# B&R Automation Studio project TD52 (part 85)

```iecst
	tLX2_Perm_aux : 	STRUCT
		iFiltConst_LeanoxDev_Gen1 : UINT; (*Filter coefficient PT1 - Leanox deviation for LX2 steady state - Gen1 [sec]*)
		rThreshold_LeanoxDev_Gen1 : REAL; (*Threshold leanox deviation for LX2 steady state - Gen1 [mbar]*)
		rThreshold_Pnorm_LX2_ramp : REAL; (*Threshold norm. power change within 1 second interval for LX2 load ramp detection [0...1]*)
		rThreshold_Pnorm_LX2_step : REAL; (*Threshold norm. power filters difference for LX2 load step detection [0...1]*)
	END_STRUCT;
	tLX2Map : 	STRUCT
		GasType : ARRAY[0..4]OF tLX2_GasType;
	END_STRUCT;
	tLX2_GasType : 	STRUCT
		rLX2_BPOC : ARRAY[0..10]OF REAL; (*actual LX2 BPOC from Permanent Storage [bar]*)
		bLX2_BPOC_measured : ARRAY[0..10]OF BOOL; (*LX2 BPOC - binary map of already measured points [true->measured]*)
	END_STRUCT;
	Pos_WG : 	STRUCT
		Exist : BOOL; (*WG position available (either CAN communication or good quality fo analog input)*)
		Act : REAL; (*WG actual position norm*)
		Set : REAL; (*WG target position norm*)
	END_STRUCT;
	WG_ActuatorState : 	STRUCT
		PosCtrl : USINT := 1; (*Position Control*)
		SelfCal : USINT := 2; (*Self Calibration*)
		Learn : USINT := 3; (*Learn*)
		WipeCycl : USINT := 5; (*Wiping Cycle*)
		Override : USINT := 6; (*Override*)
		ElFailSafe : USINT := 7; (*Electrical Failsafe*)
		ElFailSafeOv : USINT := 8; (*Electrical Failsafe then Override*)
	END_STRUCT;
	WG_StatusMSG : 	STRUCT
		Pos_Act : UINT; (*Actual Shaft Position *)
		T : INT; (*Internal Temperature range: -55 C to +195 C*)
		Pos_Set : UINT; (*Setpoint Position*)
		Fault : USINT; (*Actuator Fault*)
		State : USINT; (*Actuator State*)
		Pos_Set_Norm : REAL; (*Target Position related to Nominal*)
		Pos_Act_Norm : REAL; (*Actual Shaft Position related to Nominal*)
	END_STRUCT;
END_TYPE
```

### Modul_EngCtr.var - Package variables
```iecst
(********************************************************************
 * COPYRIGHT -- INNIO Company
 ********************************************************************
 * Package: Opstate_Pkg
 * File: module_Opstate.typ
 * Author: Mario Graus
 * Created: October 19, 2011
 ********************************************************************
 * Data types of package Opstate_Pkg
 ********************************************************************)
VAR
	IN_EC : IN_EngCtr_Struct;
	OUT_EC : OUT_EngCtr_Struct;
	ParaFactoryDefault : Para_Struct; (*First Init Values*)
	Para : Para_Struct;
	pm : Para_Struct;
	Map : Map_Struct; (* Self learning Data*)
	Cnt : Cnt_Struct; (* Self learning Data*)
	Perm : Perm_Struct; (* Permanent Data*)
	ParaEC : Gtyp_Struct;
	MM2VIS : MM2VIS_Struct;
	VIS2MM : VIS2MM_Struct;
	bEC_Trace_Trigger : BOOL; (* Trigger PV for Traces *)
	iTFilterTVref : UINT;
	iSG_PBC_GlowRed : INT;
	ucGS : USINT; (*Gas Sort (gasart)*)
	xLX2 : fLX2;
	xTrStRed : fTrStRed;
	iCntEC : USINT; (* counter variable reuseable *)
	bWG_CAN_A_Learn_On_Vis : BOOL := 0;	(*Learn On signal to VISU WG A*)
	bWG_CAN_B_Learn_On_Vis : BOOL := 0;	(*Learn On signal to VISU WG B*)
END_VAR
(* IN_EngCtr *)
VAR
	xOpMode : OpMode;
	xEngType : EngType;
	rV_EngDis : REAL; (*Engine Displacement [m3]*)
	rN_Eng : REAL; (*Engine Speed [1/min]*)
	bNewEngCycle : BOOL; (*TRUE = new engine cycle trigger*)
	bType6_Update : BOOL; (* Enables type 6 controls update*)
	bSS_PFPDR : BOOL; (* Steady State for PFPDR *)
	bSS_Opt : BOOL; (* Steady State for Optimizer*)
	bSS_LamLim : BOOL; (* Steady State for Lambda Limit*)
	bSS_WG : BOOL; (* Steady State for wastegate *)
	rH_Amb : REAL; (* Sealevel [m] *)
	rPr_Amb : REAL; (* Ambient pressure [bar] *)
	bWasActivatedGen2Idle : BOOL := FALSE;
	bIsActiveGen2Idle : BOOL := FALSE;
	rVE_Eng : REAL; (* Volumetric Efficiency *) (* OldName: rLieferGMotor; Cycle: 2 *)
	rLam_PI : REAL; (* lambda for port injection opening duration calculation *)
	xGridStat : fGridStat;
	rN_Set_Norm : REAL := 1.0; (*Speed setpoint normalized for Engine Controller*)
END_VAR
(* misf_ctr *)
VAR
	bTrip_Misf : BOOL; (* Trip: A1047 Misfiring failure *) (* OldName: AUSS_A; Cycle: 2 *)
	bWarn_Misf : BOOL; (* Warning: W3217 Misfiring failure *)
	bMisfBlink : BOOL;
	iCnt_Misf : USINT;
END_VAR
(* IgnPoint *)
VAR
	rCA_IP_Set : REAL; (* actual ignition timing setpoint *) (* OldName: W_ZZP; Cycle: 2 *)
	bSG_PBC_GlowRed : BOOL; (*Release FPR/SCO through PBC*) (* OldName: bReductionGlow_Pi; *)
	bPBC_IPRed : BOOL; (*Betriebsmeldung ZZP-Reduktion Gluehzuenden / Pmax*) (* OldName: bZZPRed_DMR; *)
	iPBC_IPRed : USINT; (*Betriebsmeldung ZZP-Reduktion Gluehzuenden / Pmax*) (* OldName: ucDMRZZPRed; *)
	iCyl_IP_Act_Min : USINT; (*Nummer vom Zylinder mit kleinsten ZZP*)
	bTrStRed_Running : BOOL; (* TrStRed function running status *)
	bTrStRed_hiEGT_dis : BOOL; (* high avg.EGT pw.red. disable / timer extension for high cyl.max.EGT alarm by TrStRed function *)
	bTrStRed_SteadyState_Loss_LX2 : BOOL; (* Leanox plus steady state loss by TrStRed function *)
	bMsg_TrStRed_Start : BOOL; (* TrStRed function cycle started - operator message *)
	bMsg_TrStRed_Complete : BOOL; (* TrStRed function cycle completed - operator message *)
	rCA_IPOffs_SCRInTemp : REAL;
END_VAR
(* dyn_GR *)
VAR
	bBM_GrC_Event : BOOL; (* Low Voltage Ride Through Event *)
	bBM_PoleSlip : BOOL; (* Mains failure + Generator Pole slip *)
	bBM_Disc_dynAng : BOOL; (* Mains failure + dynamic rotor angle maximum *)
	bBM_Disc_staticAng : BOOL; (* Mains failure + static rotor angle maximum*)
	bBM_Disc_CapMode : BOOL; (* Mains failure + leading power factor operation *)
	bBM_Disc_dynAng_Min : BOOL; (* Mains failure + dynamic rotor angle minimum *)
	bBM_Disc_Power : BOOL; (* Mains failure + electric power to low *)
	bBM_FRT_Event : BOOL; (* Fault Ride Through Event in island operation *)
	bBM_PoleSlip_EPS : BOOL; (* Generator Pole slip in island operation *)
	bBM_GrC_Event_Sim : BOOL; (* Low Voltage Ride Through Event simulated *)
	bGC_LeanoxErr_AUS : BOOL := FALSE; (*TRUE = Stoerung A1080 deaktiviert ueber GCEvent*)
	iMissfCyl_GrC : UDINT; (* 0 *) (* OldName: MissfCyl_GC; Cycle:2; *)
	bGrC_PowerFIX_HVRT : BOOL; (* TRUE = Leistungsfixierung im eng_ctr aktiv (Zeit laeuft) --> HVRT Event*) (* OldName: bGC_PowerFIX; Cycle:2; *)
	bGrC_PowerFIX : BOOL; (* TRUE = Leistungsfixierung im eng_ctr aktiv (Zeit laeuft) --> LVRT Event*) (* OldName: bGC_PowerFIX; Cycle:2; *)
	bGC_maintenance_request : BOOL; (* Mains failure maintenance request *) (* OldName: bGC_maintenance_request ; Cycle:2; *)
	bGrC_TCPumpAkt : BOOL; (* TRUE=Pumperkennung aus dyn. GC aktiv fuer gas_flow *) (* OldName: bGC_TCPumpAkt; Cycle:2; *)
	bGrC_LambAdabtAKT : BOOL; (* TURE = Lambdaadaption from dyn. GridCode aktiv *) (* OldName: bGC_LambdaAdabtAKT; Cycle:2; *)
	bVoltageLow_cust_OP_MSG : BOOL;
	bGrC_FixActuators : BOOL;
	rPos_WG_GrC : REAL;
	rPos_CBV_GrC : REAL;
	bIgnOffTestMode : BOOL := FALSE; (*TRUE = Zuendung EIN/AUS nach Muster*)
	bIGTLatePhase2ON : BOOL; (*ZZP auf spaet stellen in Phase 2 JA/NEIN*)
	bIGTLatePhase2 : BOOL; (*Befehl an ignpoint Task - ZZP auf spaet stellen*)
	rCA_Ign_Act_late_GC : REAL; (*[deg CA] spaeter ZZP fuer Phase 2 von IGNTestMode (GridCode)*)
	bFreeze_GEN2 : BOOL;
	rPos_CBV_Freeze : REAL;
	rPos_TV_Freeze : REAL;
	rPos_WG_Freeze : REAL;
	rGrid_OffsetFactor : REAL; (* PI-Duration offset from dynamic gridcode *)
	rGasflow_Factor_GrC : REAL; (* Gasflow factor from dynamic gridcode *)
	bGrC_GCB_DCON_FRT : BOOL; (* Open signal to GCB due to pole slip *)
	bGrC_GCB_DCON_FRT_EPS : BOOL; (* Open signal to GCB due to pole slip in island operation *)
	bLeanox_Man_old_FRT : BOOL; (* LEANOX controller status before FRT event *)
END_VAR
(* GR_GCB_cust *)
VAR
	bF_UnderMp_Lo : BOOL; (* W9312: Generator frequency too low in mains parallel operation *)
	bF_OverMp_Hi : BOOL; (* W9313: Generator frequency too high in mains parallel operation *)
	iTFilt_N_GR : UINT := 2000;
	rN_GR_Filt : REAL; (* Filtered engine speed for LEANOX speed compensation *)
	rF_GR_Filt : REAL; (* Filtered engine frequency for ITP reduction *)
END_VAR
(* GAS FLOW *)
VAR
	rP_Rot : REAL; (*Rotationsleistung in [kW]*)
	rLam_Trans_Corr : REAL; (*transient Lambda correction*)
	TJ_GASO : BOOL;
	TJ_GASO_B : BOOL;
	ucTJ_GASO : USINT;
	TJ_GASM : BOOL;
	TJ_GASM_B : BOOL;
	ucTJ_GASM : USINT;
	rFlow_TV_x : REAL; (*LIVC actual Volumeflow for TV Controller*)
	rFlow_TV_w : REAL; (*LIVC setpoint Volumeflow for TV Controller*)
	rFlow_CBV_x : REAL; (*LIVC actual Volumeflow for CBV Controller*)
	rFlow_CBV_w : REAL; (*LIVC setpoint Volumeflow for CBV Controller*)
	bBM2852_PumpPuls : BOOL; (*B2852 - Turbolader Pumpen*)
	rLam_TJ_Set : REAL; (* Lambda for TecJet *)
	rPr_P2s_df : REAL; (*P2s Digital gefiltert in [bar]*)
	rPr_P2s_df_TJ : REAL; (*P2s Digital gefiltert in [bar]*)
	rCBV_CDS_Speed_D_Offset : REAL; (*T6 GEN1 CBV derivative gain scheduling*)
	rTV_CDS_Speed_D_Offset : REAL; (*T6 GEN1 TV derivative gain scheduling*)
END_VAR
(* LEANOX *)
VAR
	rP_Act_l : REAL;
	rPr_Leanox_Set : REAL; (* Setpoint boost pressure *) (* Oldname: pl_soll; Cycle: 2*)
	rLam_Leanox_Set : REAL; (* Setpoint lambda *) (* Oldname: OUT_EC.rLam_Eng_LL_Set; Cycle: 2*)
	RPSW3 : BOOL; (*Warning: LEANOX algorithm failure*)
	RPSA7 : BOOL;
	rPr_CH_PFPDR_Calc : REAL; (* Boost pressure offset calculated for PFPDR*)
	rNum_ConvLamtoP2s : REAL := 2; (* Conversion rate from lambda to boost pressure for PFPDR*)
	rPr_CH_PFPDR_Offs : REAL; (* Boost pressure offset from PFPDR to Gen2 controller*)
	rCorr_LX_GR : REAL; (* Speed compensation factor for LEANOX *)
	rPr_Leanox_Offs_H2 : REAL; (* Boost pressure offset H2 content [bar] *)
END_VAR
(* eng_ctr *)
VAR
	rPos_TV_u : REAL; (*Regler Ausgang ohne skalierung*)
	iMisfCyl_OverSpeed : UDINT; (*ACHTUNG hier braucht es noch Klaerung*)
	bLR_IGN_Retard : BOOL; (*retard ignition timing point to react on a load rejection by the GCB*)
	pm_stat_var_LR : ARRAY[0..100] OF tStat_VAR_LR := [101(0)]; (*statistic structure to save the speed gradient values at engine shut down with time stamps*)
	pm_stat_var : ARRAY[0..100] OF tStat_VAR := [101((0))]; (*statistic structure to save the speed gradient values at engine shut down with time stamps*)
	iCounter_stat_var_LR : INT := 0;
	iCounter_stat_var : INT := 0; (*counter and index variable for statistic structure for the speed gradient values*)
	rN_LR_IGN_Retard_HOLD : REAL := 1.1; (*Speed threshold to keep ITP retard during LR [p.u.]*)
	rTi_LR_GasStop_largeRej : REAL := 0.4; (*Duration of gas-stop for big load rejections [s]*)
	rTi_LR_GasStop_smallRej : REAL := 0.1; (*Duration of gas-stop for small load rejections [s]*)
END_VAR
(* Msg EC *)
VAR
	bGnlTrip : BOOL;
	bGnlTrip1 : BOOL;
	bGnlTrip2 : BOOL;
	bGnlTrip3 : BOOL;
	bGnlWarning : BOOL;
	AmmSeq_PiPosAbw : AmmSequence; (* Trip: W2470, OM: B2929 *) (* Oldname: AmmSeq_PiPosAbw *)
END_VAR
(* gen_EC_T2 *)
VAR
	bAct_Mon_Release : BOOL; (*Throttle valve failure monitoring release*)
	bAct_Mon_Rel_WG : BOOL; (*Release monitoring for wastegate actuator*)
	tDataRec_EEPROM : ARRAY[0..7] OF BYTE := [8(0)]; (*CAN wastegate read data A - 8 bytes*)
	tDataRec_EEPROM_Info : ARRAY[0..7] OF BYTE := [8(0)]; (*CAN wastegate read data A - 8 bytes*)
	tCAN_WG_ADDR_A : BYTE := 0; (*CAN wastegate A source address*)
	tCAN_WG_ADDR_B : BYTE := 0; (*CAN wastegate B source address*)
	tNewADDR : BYTE := 0; (*CAN wastegate new address to configure EEPROM*)
	tWG_CAN_B_ActSrcAdd : BYTE := 0; (*CAN wastegate actuator B source address*)
	tWG_CAN_A_ActSrcAdd : BYTE := 0; (*CAN wastegate actuator A source address*)
END_VAR
(* parEC *)
VAR
	bNoInitDetected : BOOL := FALSE; (*allways true, except 1cycle on init up*)
END_VAR
(* hum_pac_EC *)
VAR
	rpl_soll_Max_filt : REAL;
	rpl_ist_filt : REAL;
	AbsHumidity : REAL; (* absolute humidity air intake [g/kg] *)
	bMsg_Hum_T2sOffs_Act : BOOL;
	bMsg_Hum_Pred_Lim : BOOL;
	pbaro : REAL; (* barometric pressure used for humidity control [bar] *)
	rP2s_Comp_HumOffset : REAL; (* [bar] *)
	rT_T2_HumOffset : REAL; (*  *)
	rMassFlow_Gas : REAL; (* gas mass flow [kg_gas/h] *)
	rMassFlow_AirIn : REAL; (* intake air mass flow [kg_air/h] *)
	AbsHumidity_Mixture : REAL; (* absolute humidity mixture [kg_H2O/kg_mix] *)
	rGasFlowN : ARRAY[0..4] OF REAL; (* gas flow [m^3/h] *)
	bHum_GasIn_Abs_MSF : BOOL; (* measuring signal failure customer signal BUS *)
	AbsHumidity_AirIn : REAL; (* absolute humidity air intake [g/kg] *)
	AbsHumidity_Mix : REAL; (* absolute humidity mixture [g/kg] *)
END_VAR
(* Exhaust *)
VAR
	AN_ABMWN : ARRAY[0..25] OF BOOL; (* Koppelfeld Abweichung neg vom Mitt*)
	AN_ABMWN_B : BOOL; (* dev. exh. avg. operating message *)
	AN_ABMWN_W : BOOL; (* negative dev. exh. avg. warning *)
	AN_ABMWP : ARRAY[0..25] OF BOOL; (* Koppelfeld Abweichung pos vom Mitt*)
	AN_ABMWP_B : BOOL; (* dev. exh. avg. operating message *)
	AN_ABMWP_W : BOOL; (* positive dev. exh. avg. warning *)
	AN_ATMA : BOOL;
	bZylAusfall : BOOL;
	bMsg1049_Test : BOOL;
	MS_AGT : BOOL;
	MSAGT : ARRAY[0..25] OF BOOL;
	MSAGT_W : BOOL;
	t_zyl : ARRAY[0..25] OF INT;
	bSCO_EGT_DltLim : BOOL; (* - *) (* OldName: AGT_DELTA; *)
	iNum_Cyl_EGT_Max : USINT; (*Hottest cylinder number*) (* OldName: ucZYL_MAX_Cyl; *)
	AN_ABMW : BOOL;
	AN_ATM : ARRAY[0..25] OF BOOL;
	MSAGT_B : BOOL;
	AN_ATMA_B : BOOL;
	rT_EG_MaxLim : REAL; (*exhaust gas temperature maximum limit*)
	xTExhMon : fTExhMon := (0); (*FuB*)
	bMsg2339_Set : BOOL; (* A2339: Exhaust gas temperature inclination maximum at cylinder head *)
	bMsg2970_Set : BOOL; (* B2970: Exhaust gas temperature inclination maximum at cylinder head *)
	iNum_Msg2970 : USINT;
	bHoldBackfPrev : BOOL;
	bMsg9388_Set : BOOL; (*W9388: Combustion anomaly detected*)
	bMsg9092_Set : BOOL; (*B9092: Combustion anomaly detected*)
END_VAR
(* GLOW IGN *)
VAR
	bSG_TV : BOOL; (*Enables TV alternation by GlowIgnition Task*)
	rPos_SG_TV : REAL; (*alternated TV postion*)
	bSG_CBV : BOOL; (*Enables CBV alternation by GlowIgnition Task*)
	rPos_SG_CBV : REAL; (*alternated CBV position*)
	bSG_Rel_Mon : BOOL; (* monitoring release for special gas applikation *) (* Oldname: FG_TS_UW *)
	bSCO_BLOCK1 : BOOL; (* Blockierung Sicherheitsschliessen *) (* OldName: SS_BLOCK1; *)
	bSCO_BLOCK2 : BOOL; (* Blockierung Sicherheitsschliessen *) (* OldName: SS_BLOCK2; *)
	bSG_PBC_GlowIgnFailure : BOOL; (* Glow ignition failure by PBC *) (* OldName: bDMR_A_GLOW; *)
	rSG_GasLimit : REAL; (* special gas factor for gasflow limit *) (* OldName: ssGasLimit; *)
	bSG_BackFireDetection : BOOL; (* Trip A2283 *)
	bSG_TV_FGQC : BOOL; (* Fix TV position *)
	bSG_CBV_FGQC : BOOL; (* Fix CBV position *)
	rPos_SG_TV_FGQC : REAL; (* TV position FGCQ *)
	rPos_SG_CBV_FGQC : REAL; (* CBV position FGCQ *)
	b2975_Set : BOOL; (* Operation message 2975 *)
	bFGQC_Active : BOOL; (* Fast gas quality change function active *)
	bLeanox_Man_oldFGQC : BOOL; (* LEANOX controller status before FGQC event *)
	bFPR_Active : BOOL; (* Fast power reduction function active *)
	bLeanox_Man_old_FPR : BOOL; (* LEANOX controller status before FPT event *)
END_VAR
(* PFPDR *)
VAR
	rLam_PFPDR_Offs : REAL; (* Lambda Offset during PFPDR *)
	bPFPDR_IPCorr_dis : BOOL; (* disables IP correction during PFPDR *)
	rCA_IP_PFPDR_Offs : REAL;
	bPFPDR_CylOpt_dis : BOOL;
	bPFPDR_CBVOpt_dis : BOOL;
	bPFPDR_Act : BOOL;
	bIP_CBVOpt : BOOL; (* CBVOpt aktiv? *)
	rCA_IP_PFPDR_Prof : ARRAY[0..24] OF REAL;
	MFB50Ctr : AI50toIT;
	bTrace_var : BOOL := 0;
	rCA_MFB50_Filt_type9 : ARRAY[0..24] OF REAL;
	rCA_MFB50_Filt_type6_Max : REAL;
	rCA_MFB50_Filt_type6_Min : REAL;
	rCA_MFB50_Filt_type6_Avg : REAL;
	rCA_MFB50_Filt_type6 : ARRAY[0..24] OF REAL;
	rCA_MFB50_Filt_type6_Median : REAL;
	rCA_MFB50_Filt_type9_Median : REAL;
	rCA_MFB50_type9_Set : REAL;
	rCA_MFB50_Filt_type9_Min : REAL;
	rCA_MFB50_Filt_type9_Max : REAL;
	rCA_MFB50_Filt_type9_Avg : REAL;
	rCA_MFB50_type6_Set : REAL;
	rPr_Leanox_Offset_CoV : REAL;
	rPos_TB34_SG : REAL;
	iTB34CtrMode : INT;
	bTrip_LambdaLimit : BOOL; (*A2294: Lambda limit exceeded*)
	bMsg_p2soutofRange : BOOL; (*B2897: Boost pressure out of range*)
	bGEN2_Block_P2_Err : BOOL; (* Block Gen2: no P2 pressure signal available *)
	xGen2 : Gen2;
	bGEN2_FDC_active : BOOL; (*Activate Hangs FDC in GEN2 control*)
	bVerrigelung_EXHT : BOOL;
	refPoint_Lambda_start : ARRAY[0..9] OF lcrCurveByPoints_TabEntry_type;
	LCRCByP_Lambda_start : LCRCurveByPoints;
	refPoint_ITP : ARRAY[0..9] OF lcrCurveByPoints_TabEntry_type;
	LCRCByP_ITP : LCRCurveByPoints;
	refPoint_LamLoLim_coldFS_ABS : ARRAY[0..9] OF lcrCurveByPoints_TabEntry_type; (* y = abs lam limit and x = pressure in [bar] *)
	refPoint_LamLoLim_ABS : ARRAY[0..9] OF lcrCurveByPoints_TabEntry_type; (* y = abs lam limit and x = pressure in [bar] *)
	refPoint_LamUpLim_ABS : ARRAY[0..9] OF lcrCurveByPoints_TabEntry_type; (* y = abs upper lam limit and x = pressure in [bar] *)
	rZZPStart_T4_low : REAL;
	rZZPStart_T4_high : REAL;
	bITPStTEMP : BOOL;
	bFirstStepAct : BOOL;
	bExhTempDep : BOOL;
	rFirstStepITPOffs : REAL;
	rSecondStepITPOffs : REAL;
	rCA_IT_GEN2_FS_rel : REAL;
	ulGasFlow_M_FDC : UDINT; (*[Nl/s] * 1000*)
	ulGasFlow_FDC : UDINT; (*[Nl/s] * 1000*)
	rN_StartITOffs_full : REAL;
	rN_StartITOffs_zero : REAL;
	rCA_IP_Set_Raw_GEN2_FS : REAL;
	rP_IT_FS_LimNorm : REAL;
	tmaxITP : TIME;
	rCA_IT_Offs_Start : REAL;
	rCA_IP_Gen2_Offs : REAL;
	rCA_IP_Gen2_NetP_Offs : REAL;
	bGEN2_FS_IP_Set : BOOL := 0;
	rZZPStart_Tcyl_low : REAL := 0;
	rZZPStart_Tcyl_high : REAL := 0;
	rCA_IP_Set_Raw_normal : REAL;
	rT_EG_H : ARRAY[0..24] OF REAL;
	TP_10ms_OptiChng : TP_10ms := (0);
	iCount_steady : INT;
	iNum_steady_state : INT;
	bdeltaPr_TV_actuateTV : BOOL;
	rGainTV_rDeltaPr_TV : REAL;
	rDeltaPr_TV_integrator_TV : REAL;
	rDeltaPr_TV_integrate_TV_ON : REAL;
	rPr_CBV_Release : REAL;
	rPr_CBV_Lock : REAL;
	deltaPr_TV_ref_data : ARRAY[0..5] OF lcrCurveByPoints_TabEntry_type;
	deltaPr_TV_CBV_gain_data : ARRAY[0..5] OF lcrCurveByPoints_TabEntry_type;
	deltaPr_TV_TV_gain_data : ARRAY[0..5] OF lcrCurveByPoints_TabEntry_type;
	CBV_lim_byTV_data : ARRAY[0..4] OF lcrCurveByPoints_TabEntry_type;
	LCRCurve_TV_min_table : ARRAY[0..7] OF lcrCurveByPoints_TabEntry_type;
	LCRCurve_TV_min_CBV_table : ARRAY[0..2] OF lcrCurveByPoints_TabEntry_type;
	rP_LR_Trig_ActSat_CBV : REAL;
	rTi_LR_ActSat_CBV : REAL;
	xLCRCurve_R_Rot_Correction_data : ARRAY[0..8] OF lcrCurveByPoints_TabEntry_type;
	rDelta_a_red : REAL := 0.0;
	bSIMPID_EXT_TV_Act : BOOL := FALSE;
	bSIMPID_EXTERN_AW_TV : BOOL := FALSE;
	bSIMPID_EXTERN_AW_CBV : BOOL := FALSE;
	bSTOPint_cbv_trans : BOOL := FALSE;
	rP_el_LockTV_Norm : REAL; (*Power trigger value to lock the throttle valve in island mode in upper load range*)
	rP_el_ReleaseTV_Norm : REAL; (*Power trigger value to release the throttle valve in island mode*)
	tTimeTrigger : TIME := T#150ms;
	tTimeTrigger_HiGasDens : TIME := T#60ms;
	ulGasSprungVol : UDINT; (*[l/s]*1000*)
	ulGasSprungVol_HiGasDens : UDINT; (*[l/s]*1000*)
	bstveract : BOOL;
	bGasSprung : BOOL;
	ulatvergasvol : UDINT;
	ulGasSprungMax : UDINT; (*[l/s]*1000*)
	iGasSprungThresh_HiGasDens : INT; (*[g/Nm3]*)
	bUseTVIdleControl : BOOL; (*TRUE = Engine uses TV control without skipfire for engine start and idle control*)
	rKp_Gen2SkipF_Pnom : REAL;
	rKp_Gen2SkipF_Pskip : REAL;
	rP_LimitBDCCBV_ff_Active : REAL;
END_VAR
(*LeanoxDrift*)
VAR
	bWarn_Nox_Meas_recommend : BOOL; (*warning for recommend leanox adjustment*)
	bWarn_Nox_Meas_mandatory : BOOL; (*warning for mandatory leanox adjustment*)
	bMsg_B2937 : BOOL; (*B2937: operating message for performed leanox adjustment*)
	bMsg_B2938 : BOOL; (*B2938: operating message for performed combustion chamber cleaning*)
	bCBV_closed_Start_SY : BOOL; (*TRUE = CBV closed at engine start until SY*)
	bParaSetupOk_10s : BOOL; (*Para Setup OK + 10sec*)
	bFS_Ramp_Rel : BOOL;
	bTiStart5min_Ena : BOOL;
	bEngine_was_stopped : BOOL := 0;
	rF_LEANOX_Err : REAL := 1.0;
	bGEN2_RAMP_ACTIVE : BOOL := 0;
	bUseColdFS_LamLim : BOOL := 0; (*Use cold Fast Start low Lambda Limits for GEN2*)
	bMisfGEN2 : BOOL := TRUE; (*activate misfire computed from GEN2 control*)
	iMissfCyl_GEN2 : UDINT := 0; (*number of skipped cylinders from GEN2 control*)
	refPoint_addKpLam_Kp_y : ARRAY[0..5] OF REAL; (*reference add Lambda Kp GEN2 island*)
	rKeAdaptRL : REAL; (*reference gain for adaption GEN2 island*)
	rKeAdaptGain : REAL; (*reference rate limit for adaption GEN2 island*)
	rITCtransDeltaAcc_y : ARRAY[0..4] OF REAL; (*reference for transient ignitioin timing point change of GEN2 to avoid knocking*)
	refPoint_iLQR_Q0_y : ARRAY[0..5] OF REAL; (*reference Q0 GEN2 island*)
	refPoint_addKpLam_Ti_y : ARRAY[0..5] OF REAL; (*reference add Lambda Ti GEN2 island*)
	refPoint_iLQR_Keng_y_pow : ARRAY[0..6] OF REAL; (*reference to reset learning function*)
	refPoint_iLQR_Keng_y : ARRAY[0..12] OF REAL; (*reference to reset learning function*)
	bdcCbv_rKp_island_Lup : ARRAY[0..9] OF REAL; (*reference gain scheduling Kp bypass valve for GEN2 BDC island*)
	bdcTv_rKp_island_Lup : ARRAY[0..9] OF REAL; (*reference gain scheduling Kp throttle valve for GEN2 BDC island*)
	refPoint_iLQR_R1_y : ARRAY[0..5] OF REAL; (*reference R1 GEN2 island*)
	bAutoLoad_Island : BOOL; (*Werte fuer GEN2 Inselbetrieb laden in PV-CHECK*)
END_VAR
(* ESC *)
VAR
	rLamLimOffs_ESC : REAL; (* Lambda lower limit offset ESC *)
	rP_Ramp_IncGrad_Offs_ESC : REAL; (* Power ramp offset ESC *)
END_VAR
(*Leanox 2.0*)
VAR
	bLX2_active : BOOL; (*Leanox 2.0 active [true->active]*)
	bWarn_LX2_inLimit : BOOL; (*Leanox 2 saturation - warning*)
	bMsg_LX2_Active : BOOL; (*Leanox 2 Active - operator message*)
	bMsg_LX2_NotActive : BOOL; (*Leanox 2 Not Active - operator message*)
	bMsg_LX2_MapReset : BOOL; (*Leanox 2 Map Reset Request from HMI - operator message*)
	rMFIntOutMax : REAL; (*Misfire level used for ESC and LX2*)
	rPr_LX2_offset : REAL; (* Leanox 2.0 boost pressure offset *)
	rGain_ss_boost_iLQR : REAL := 0.0;
	rGain_ss_boost_iLQR_OUT : REAL := 0.0;
	bDemPermSave : BOOL;
END_VAR
(* FastStart *)
VAR
	bLoad_reached : BOOL;
	bTarLoad_reached : BOOL;
	bTarLoad_blockOM : BOOL;
	xTP_TarLoad_reached : TP;
	bFS_Island_Ena : BOOL; (* island fast start enabled *)
END_VAR
(* Direct Air Injection *)
VAR
	xDAI : fDAI; (* direct air injection FB *)
	bDAI_MSF : BOOL; (* direct air injection measuring signal failure *)
	bDAI_V_Close_Fault : BOOL; (* direct air injection shut off valve closing fault *)
	bDAI_V_Open_Fault : BOOL; (* direct air injection shut off valve opening fault *)
	bDAI_Pr_In_Hi : BOOL; (* direct air injection pressure before shut off valve high *)
	TOF_MissfCmd : TOF;
END_VAR
(* TC1 SPP *)
VAR
	rPr_EGbHP_TC1 : tBank_AB; (* P3 Filt TC1*)
	rPr_EGbHP_TC1_UF : REAL;
END_VAR
(* TC2 SPP_EC *)
VAR
	bT_SCR_OXI_TC_valid : BOOL; (*Inlet temperature sensor exist and good quality - SCR in, SCR out, OXIcat In, Turbocharger Out*)
	rT_SCR_OXI_TC_In_Hi : REAL; (*Inlet temperature maximum - SCR in, SCR out, OXIcat In, Turbocharger Out [degC]*)
END_VAR
(* Wastegate *)
VAR
	rPos_CBV_Ref_WG : REAL; (*setpoint of position compressor bypass valve for wastegate control*)
	rPosWG_Factor : REAL := 0.0; (*CAN wastegate read position factor*)
	tDataSend_WG : ARRAY[0..7] OF BYTE := [8(0)]; (*CAN wastegate data to send - 8 bytes*)
	iDataSend_WG_Tmp : UINT := 0; (*CAN wastegate set position to be sent - TEMPORARY*)
	tDataSend_WG_Tmp : ARRAY[0..1] OF BYTE := [2(0)]; (*CAN wastegate actuator command TEMPORARY byte*)
	iCAN_WG_B_StatID : ARRAY[0..5] OF UDINT := [6(0)]; (*CAN wastegate actuator B - Actuator Status MSG ID*)
	iCAN_WG_B_ErrID : ARRAY[0..5] OF UDINT := [6(0)]; (*CAN wastegate actuator B - Failures and Warning MSG ID*)
	iCAN_WG_B_SendID : ARRAY[0..5] OF UDINT := [6(0)]; (*CAN wastegate actuator B - Actuator Command MSG ID*)
	iCAN_WG_A_StatID : ARRAY[0..5] OF UDINT := [6(0)]; (*CAN wastegate actuator A - Actuator Status MSG ID*)
	iCAN_WG_A_ErrID : ARRAY[0..5] OF UDINT := [6(0)]; (*CAN wastegate actuator A - Failures and Warning MSG ID*)
	iCAN_WG_A_SendID : ARRAY[0..5] OF UDINT := [6(0)]; (*CAN wastegate actuator A - Actuator Command MSG ID*)
	iCAN_WG_A_T2AID : ARRAY[0..5] OF UDINT := [6(0)]; (*CAN wastegate actuator A - Tool to Actuator MSG ID*)
	iCAN_WG_A_A2TID : ARRAY[0..5] OF UDINT := [6(0)]; (*CAN wastegate actuator A - Actuator to Tool  MSG ID*)
	iCAN_WG_B_T2AID : ARRAY[0..5] OF UDINT := [6(0)]; (*CAN wastegate actuator B - Tool to Actuator MSG ID*)
	iCAN_WG_B_A2TID : ARRAY[0..5] OF UDINT := [6(0)]; (*CAN wastegate actuator B - Actuator to Tool  MSG ID*)
	iCAN_WG_DataLength : ARRAY[0..5] OF USINT := [6(0)]; (*CAN wastegate data length (K_S: 8 bytes)*)
	xCANread_WG_B_EE : CANread := (0); (*CAN wastegate B read function*)
	xCANread_WG_A_EE : CANread := (0); (*CAN wastegate A read function*)
	xCANwrite_WG_B_EE : CANwrite := (0); (*CAN wastegate B write function*)
	xCANwrite_WG_A_EE : CANwrite := (0); (*CAN wastegate A write function*)
	xCANreadID_WG : CANread := (0); (*CAN wastegate A/B ID read function*)
	xCANwrite_WG_B : CANwrite := (0); (*CAN wastegate B write function*)
	xCANwrite_WG_A : CANwrite := (0); (*CAN wastegate A write function*)
	xCANwriteID_WG_B : CANwrite := (0); (*CAN wastegate B write function*)
	xCANwriteID_WG_A : CANwrite := (0); (*CAN wastegate A write function*)
	xCANread_WG_B : CANread := (0); (*CAN wastegate B read function*)
	xCANread_WG_A : CANread := (0); (*CAN wastegate A read function*)
	iWG_CAN_A_State : USINT := 0; (*CAN wastegate actuator A commanded state*)
	iWG_CAN_B_State : USINT := 0; (*CAN wastegate actuator B commanded state*)
	tPos_WG_A : Pos_WG := (0); (*Wastegate position actuator A*)
	tPos_WG_B : Pos_WG := (0); (*Wastegate position actuator B*)
	tPos_WG : Pos_WG := (0); (*Wastegate position actuator single*)
	bActuator_WG_A_Exist : BOOL := FALSE; (*Wastegate actuator A exists*)
	bActuator_WG_B_Exist : BOOL := FALSE; (*Wastegate actuator B exists*)
	bActuator_WG_Exist : BOOL := FALSE; (*Wastegate actuator single exists*)
	bActuator_WG_A_Ok : BOOL := FALSE; (*Wastegate actuator A is OK*)
	bActuator_WG_B_Ok : BOOL := FALSE; (*Wastegate actuator B is OK*)
	bActuator_WG_Ok : BOOL := FALSE; (*Wastegate actuator single *)
	tWG_CAN_A_Warn : ARRAY[0..1] OF BYTE := [2(0)]; (*CAN wastegate A System Warnings*)
	tWG_CAN_A_Fail : BYTE := 0; (*CAN wastegate A Actuator Failures*)
	tWG_CAN_B_Warn : ARRAY[0..1] OF BYTE := [2(0)]; (*CAN wastegate B System Warnings*)
	tWG_CAN_B_Fail : BYTE := 0; (*CAN wastegate B Actuator Failures*)
	bErr_WG_CANcomm_A : BOOL := 0; (*CAN wastegate A CAN communication A2384 set*)
	bErr_WG_CANfail_A : BOOL := 0; (*CAN wastegate A CAN failures W2380 set*)
	bErr_WG_CANwarn_A : BOOL := 0; (*CAN wastegate A CAN warnings W2382 set*)
	bErr_WG_CANcomm_B : BOOL := 0; (*CAN wastegate B CAN communication A2385 set*)
	bErr_WG_CANfail_B : BOOL := 0; (*CAN wastegate B CAN failures W2381 set*)
	bErr_WG_CANwarn_B : BOOL := 0; (*CAN wastegate B CAN warnings W2383 set*)
END_VAR
VAR CONSTANT
	tWG_ActuatorState : WG_ActuatorState := (PosCtrl:=1,SelfCal:=2,Learn:=3,WipeCycl:=5,Override:=6,ElFailSafe:=7,ElFailSafeOv:=8); (*CAN wastegate actuator K&S: available commanded states*)
END_VAR
VAR
	tWG_A_Status : WG_StatusMSG; (*CAN wastegate A CAN Status Information*)
	tWG_B_Status : WG_StatusMSG; (*CAN wastegate B CAN Status Information*)
	bCANread_WG_A_Err : BOOL; (*CAN wastegate A CAN read error trigger bit*)
	bCANread_WG_B_Err : BOOL; (*CAN wastegate B CAN read error trigger bit*)
END_VAR
(* PCGV Monitoring *)
VAR
	xPCGVmon : fPCGVmon; (*FuB PCGV monitoring*)
END_VAR
(* FastSync *)
VAR
	xFSyPrM : fFSyPrM; (* FastSync controller for premixed engines *)
	rPos_TV_FSyOffset : REAL := 0.02; (*TV offset when FastSync controller (premixed) is active*)
	rLam_FSyPrM_Offset : REAL := 0.0; (*Lambda offset by FastSync controller for premixed engines*)
	bFSync_StartFrom0rpm : BOOL := FALSE; (* Fast-sync w. PI: release FastSync controller only at first synchronization, engine starting from standstill*)
	bFSyPrM_StartFrom0rpm : BOOL := FALSE; (* Fast-sync premixed: release FastSync controller only at first synchronization, engine starting from standstill*)
END_VAR
(* Gen2_xt *)
VAR
	refPoint_rEtaBrakeExt : ARRAY[0..5] OF lcrCurveByPoints_TabEntry_type;
	refPoint_rGain_iLQR_rR0 : ARRAY[0..1] OF lcrCurveByPoints_TabEntry_type; (* gain for R0 value *)
	rR0_iLQR : LREAL; (*iLQR spur of R matrix *)
	rPrR_deltaP_TV_x_2 : REAL;
	rPrP2s_GEN2GQCOffs_maxLoLoad : REAL; (*[mbar] maximum GEN2 gasquality change boost pressure offset w/o scaling Parameter*)
	rR_iLQR_0 : REAL := 5.0; (* GEN2 island T6PreM *)
	rR_iLQR_1 : REAL := 40.0; (* GEN2 island T6PreM *)
	rR_iLQR_2 : REAL := 1000000000; (* GEN2 island T6PreM *)
	rR_iLQR_3 : REAL := 1000000000; (* GEN2 island T6PreM *)
	rQ_iLQR_0 : REAL := 1.0; (* GEN2 island T6PreM *)
	rQ_iLQR_1 : REAL := 0.1; (* GEN2 island T6PreM *)
	rQ_iLQR_2 : REAL := 0.0001; (* GEN2 island T6PreM *)
	rP_1_SkipF_Fact : REAL; (* Factor for 0 cylinder skipping power threshold [%Pnom] *)
	refPoint_SkipFLevel : ARRAY[0..4] OF lcrCurveByPoints_TabEntry_type; (* scaling of skip fire level over boost pressure *)
	rQ_KF_3_init : REAL := 0.01;
	rN_ssTVdpCtrl_0 : REAL := 10.0;
	rPr_delta_p2s_resetTVdp_0 : REAL := 0.5;
END_VAR
(* skip_zde *)
VAR
	iSkipF_SCRTCtr : INT; (* skip firing cylinders from SCR inlet temperature controller *)
	bSCRTCtr_SkipF_active : BOOL; (* skip fire from SCR inlet temperature controller active *)
	rT_SCRTCtr : REAL; (* SCR inlet temperature controller input *)
END_VAR
(* PVCheckNew *)
VAR
	bPermFailed : ARRAY[0..24] OF BOOL; (* Bits for Engine Block due to calibration load failure  *)
	bPermFailedComb : ARRAY[0..24] OF BOOL; (*Bits for Engine Block due to calibration load failure PVCheck and PVCheckNew combined  *)
	tOM_EngineBlocked : AmmSequence; (*OM: B2894, Engine map is missing*)
	bTrip_PoleSlip : BOOL := 0; (*Trip due to too many pole slip events*)
	xLCRCurve_Lam_Adapt_Offs_tab : ARRAY[0..10] OF lcrCurveByPoints_TabEntry_type; (*T6 GEN1 island controller lambda adaption offset map*)
	bT6_StdbyVersion : BOOL := 0; (*Activation of J6xxJ78x standby version features*)
END_VAR
(* gassort_int *)
VAR
	rCA_IgnP_Offs_H2 : REAL; (* ITP offset via H2 [deg.CA] *)
END_VAR
```

### Modul_EngCtr_Type9.var - Package variables
```iecst
(********************************************************************
 * COPYRIGHT --
 ********************************************************************
 * Package: EngineController
 * File: Modul_EngCtr_Type9.var
 * Author: Michael
 * Created: February 18, 2014
 ********************************************************************
 * Variables of package EngineController
 ********************************************************************)
(* PBC *)
VAR
	bCPP_DevLim_Underrun : ARRAY[0..24] OF BOOL; (*global an ign point übergen*) (* OldName: bPmaxLimitUntes; Cycle: 2 *)
	bCPP_DevLim_Overrun : ARRAY[0..24] OF BOOL; (*global an ign point übergen*) (* OldName: bPmaxLimitUebers; Cycle: 2 *)
	iCnt_Misf_IMEP_Max : USINT; (* IMEP Misfire Counter *) (* OldName: auss_count_PiMx; Cycle: 2 *)
	tTrip_CPP_AbsLim : AmmSequence; (* Trip: A2262, OM: B2826, Cylinder peak pressure high *) (* OldName: bAPmaxAbsLimit, bBPmaxAbsLimit, ucPmaxAbsLimit; Cycle: 2 *)
	bTrip_CPP_AvgLim : BOOL; (* Trip: A2282 average cylinder peak pressure maximum *) (* OldName: bPmax_MW_max; Cycle: 2 *)
	tTrip_CPP_DevLim : AmmSequence; (* Trip: A2274, OM: B2808, Cylinder Information *) (* OldName: bAPmaxLimit, bBPmaxLimit, ucPmaxLimit; Cycle: 2 *)
	tWarn_CPP_AbsLim : AmmSequence; (* Warning: W2588, OM: B2825, Cylinder Information *) (* OldName: bAPmaxWarnung, bBPmaxWarnung, ucPmaxWarnung; Cycle: 2 *)
	bPBC_Active : BOOL; (* PBC is active, since activation power is reached *)
	refPoint_PwrCtrKi : ARRAY[0..2] OF lcrCurveByPoints_TabEntry_type;
	tOM_CppInt_IgnRed : AmmSequence; (* Operation Msg: B2960, Cylinder Peak Pressure Integrator Iginition timing reduction *)
END_VAR
(* PI CTR and PI BAL - Port Injection Control and Balancing *)
VAR
	tOM_PI_Dur_Lim : AmmSequence; (* OM: Bxxxx, Port Injection duration limit reached*) (* OldName: bAPIDuration_HIGH, bBPIDuration_HIGH, ucPIDuration_HIGH; Cycle: 2 *)
	tWarn_PI_Dur_High : AmmSequence; (* Warn: W9216, OM: B2814, Port Injection duration is too high *) (* OldName: bAPIDuration_HIGH, bBPIDuration_HIGH, ucPIDuration_HIGH; Cycle: 2 *)
	rCA_PI_Dur_SOffset : ARRAY[0..24] OF REAL; (* sum PI duration offset: pi_bal --> pi_ctr *) (* OldName: ssSummenOffsetDuration; Cycle: 2 *)
	rCA_PI_Duration : REAL; (* global PI duration *) (* OldName: rPI_Duration; Cycle: 2 *)
	rV_CylDisp : REAL; (* Engine displaced volume *) (* OldName: rHubVolumen; Cycle: 2 *)
	rLam_PI_Set : REAL; (* Lambda for PortInjection *)
	rCA_PI_Dur_Avg : REAL; (* PI duration average*)
	rCA_PI_Dur_Min : REAL; (* PI duration minimum*)
	rCA_PI_Dur_Max : REAL; (* PI duration maximum*)
	rCA_PI_Dur : ARRAY[0..24] OF REAL; (* PI duration *)
	bOM_PI_ResetMap : BOOL; (* OM: B3235, Port injection balancer map deleted *) (* OldName: bBM_bResetMap; Cycle: 2 *)
	bOM_PI_SaveMap : BOOL; (* OM: B3236, Port injection balancer map stored *) (* OldName: bBM_bMapSave; Cycle: 2 *)
	bSteadyState_Bal : BOOL;
	bOM_PI_CommModeOn : BOOL; (* OM: B2187, Comm Mode activated *) (* OldName: newPV; Cycle: 2 *)
	bOM_PI_CommModeOff : BOOL; (* OM: B2188, Comm Mode deactivated *) (* OldName: newPV; Cycle: 2 *)
	bOM_PI_SaveToMap : BOOL; (* OM: B1299, Optimizer Map altered *) (* OldName: newPV; Cycle: 2 *)
	bFreeze_Ena_Knck : BOOL; (* enables freezing due knock, if cyls are not frozen due knock then pmax offset correction is done *)
	bLamLim_Thrs : BOOL; (* Low lambda limit threshold reached *)
	rPr_P2s_lim : REAL := 2.000;
	tOM_PI_Dur_Opt_total_Lim : AmmSequence; (* total duration offset (+map) from optimizer is in limitation *)
	tOM_PI_Dur_Opt_com_blocked : AmmSequence; (* mapping is locked by FAR detection of individual cylinders *)
END_VAR
(* SPP_EC - Signal Pre-Processing *)
VAR
	rPr_GRail_fast : REAL; (* filtered Gas rail pressure*) (* OldName: new; Cycle: 2 *)
	rPr_GRail : REAL; (* filtered Gas rail pressure*) (* OldName: new; Cycle: 2 *)
	rPr_P2s_Opt : REAL; (* filtered P2s for optimizer*) (* OldName: new; Cycle: 2 *)
	rPr_P2s_fast : REAL; (* filtered P2s *) (* OldName: new; Cycle: 2 *)
	rPr_P2s : REAL; (* filtered P2s *) (* OldName: new; Cycle: 2 *)
	rPr_P2s_A : REAL; (* filtered P2s Channel A *) (* OldName: ssPressP2s_A and rPressP2_A; Cycle: 2 *)
	rPr_P2s_B : REAL; (* filtered P2s Channel B *) (* OldName: ssPressP2s_B and rPressP2_B; Cycle: 2 *)
	rPr_P2s_UF : REAL; (* unfiltered P2s *) (* OldName: ssPressP2s_AVG; Cycle: 2 *)
	rPr_P2s_A_UF : REAL; (* unfiltered P2s Channel A *) (* OldName: rPr_Ch_P2s_A; Cycle: 2 *)
	rPr_P2s_B_UF : REAL; (* unfiltered P2s Channel B *) (* OldName: rPr_Ch_P2s_B; Cycle: 2 *)
	rPr_EGbHPTC : REAL; (* Exhaust gas pressure before high-pressure turbocharger *)
	rPr_EGbHPTC_UF : REAL; (* Exhaust gas pressure before high-pressure turbocharger unfiltered*)
	rT_T2s : REAL; (* limited T2s *) (* OldName: new; Cycle: 2 *)
	rT_T2s_A : REAL; (* limited T2s Channel A *) (* OldName: rT_Ch_T2s_A; Cycle: 2 *)
	rT_T2s_B : REAL; (* limited T2s Channel B *) (* OldName: rT_Ch_T2s_B; Cycle: 2 *)
	rT_GRail : REAL; (* limited gas rail temperature *) (* OldName: rGRTP; Cycle: 2 *)
	rCA_CPP : ARRAY[0..24] OF REAL; (* position of cylinder peak pressure *) (* OldName: ssPmaxPos; Cycle: 2 *)
	rPr_CPP_Filt : ARRAY[0..24] OF REAL; (* cylinder peak pressure filtred containment V3*) (* OldName: DruckMax; Cycle: 2 *)
	rPr_CPP : ARRAY[0..24] OF REAL; (* cylinder peak pressure *) (* OldName: DruckMax; Cycle: 2 *)
	rPr_49bfTDC : ARRAY[0..24] OF REAL; (* cylinder pressure 49° before TDC *) (* OldName: rP_49bfTDC; Cycle: 2 *)
	rPr_49afTDC : ARRAY[0..24] OF REAL; (* cylinder pressure 49° after TDC *) (* OldName: rP_49afTDC; Cycle: 2 *)
	rPr_Knck : ARRAY[0..24] OF REAL; (* knock pressure *) (* OldName: Klopfen; Cycle: 2 *)
	rPr_IMEP : ARRAY[0..24] OF REAL; (* Indicated Mean Effective Pressure *) (* OldName: IndiMitDr; Cycle: 2 *)
	rPr_ILCP : ARRAY[0..24] OF REAL; (* Indicated Load Change Pressure *) (* OldName: IndiLwDr; Cycle: 2 *)
	rCA_MFB10 : ARRAY[0..24] OF REAL; (* 10% of fuel mass burned *) (* OldName: usUmstzpkt10P; Cycle: 2 *)
	rCA_MFBvar : ARRAY[0..24] OF REAL; (* 50% of fuel mass burned *) (* OldName: UmsatzpunktL; Cycle: 2 *)
	rCA_MFB90 : ARRAY[0..24] OF REAL; (* 90% of fuel mass burned *) (* OldName: usUmstzpkt90P; Cycle: 2 *)
	rN_DMR : ARRAY[0..24] OF REAL; (* actual engine speed from DMR *) (* OldName: n_ist_DMR; Cycle: 2 *)
	bGlowIgn : ARRAY[0..24] OF BOOL; (* glow ignition *) (* OldName: Gluehzuend; Cycle: 2 *)
	bMisf_I : ARRAY[0..24] OF BOOL; (* missfire detection 10° after TDC *) (* OldName: Aussetzer; Cycle: 2 *)
	bMisf_II : ARRAY[0..24] OF BOOL; (* missfire detection 40° after TDC *) (* OldName: Misf_II; Cycle: 2 *)
	tRealTime : rtctime_typ; (* time structure *) (* OldName: new PV; Cycle: 2 *)
	iSort_Cyl : ARRAY[0..24] OF USINT; (* cylinder sorted by exhaust gas temperature *)
	rT_EG_Med : REAL; (* median of exhaust gas temperature *)
	rT_EG_MedDlt : ARRAY[0..24] OF REAL; (* exhaust gas temperature delta to median *)
	rT_EG_AvgDlt : ARRAY[0..24] OF REAL; (* exhaust gas temperature delta to average *)
END_VAR
(* PUSL - Power Unit Safety Layer *)
VAR
	tOM_MisfFail : AmmSequence; (* OM: B2849, Misfiring failure PBC *)
	iNum_HiCtr_SkipCyl : INT; (* Number of skipping cylinders from High controller*) (* OldName: ssHiGlobEng_SkipCylNr; Cycle: 2 *)
	bTrip_MaxMisfShutDown : BOOL; (* A2287 Shutdown by hierarchic controller (Misf Prio2) *) (* OldName: newPV; Cycle: 2 *)
	bTrip_MisfShutDown : BOOL; (* A2287 Shutdown by hierarchic controller (Misf Prio3) *) (* OldName: bTripPrio3_Misf; Cycle: 2 *)
	bWarn_MisfShutDown : BOOL; (* W2583 Shutdown by hierarchic controller in X min *)
	ti_MisfShutDown : TIME; (* Time until shutdown from Misfire controller *)
	bTrip_HiCtrShutDown : BOOL; (* A2287 Shutdown by hierarchic controller *) (* OldName: bHiGlobEng_EngShutDwn; Cycle: 2 *)
	bTrip_PBCSigErrFT : BOOL; (* A2290 Cylinder pressure sensor measuring signal failure *) (* OldName: bAPBCSigErrFT; Cycle: 2 *)
	tTrip_PBCSigErr : AmmSequence; (* Trip: A2290, OM: B2874, Safety layer sensor failure *) (* OldName: bAPBCSigErr, bBPBCSigErr, ucPBCSigErr; Cycle: 2 *)
	tWarn_PBCSigErr : AmmSequence; (* Warn: W2577, OM: B2802, Cylinder pressure sensor measuring signal failure *) (* OldName: bAPBCSigErr, bBPBCSigErr, ucPBCSigErr; Cycle: 2 *)
	bHiCtr_Leanox_Ena : BOOL; (* Enable high control leanox correction *) (* OldName: bLeanox_HierarchyCont; Cycle: 2 *)
	rHiCtr_Leanox_Corr : REAL; (* High control leanox correction *) (* OldName: rHiGlobEng_LEANOXCor; Cycle: 2 *)
	rHiCtr_PI_Dur_Offs : ARRAY[0..24] OF REAL; (* Duration Offset HiCtr in % *) (* OldName: rHiContrCyl_PIDUROffsetCyl; Cycle: 2 *)
	rHiCtr_PMax_Offs_Intgr : ARRAY[0..24] OF REAL; (* High Controller Pmax offset integrator *) (* OldName: rPMaxOffset_int; Cycle: 2 *)
	bLimpHomeCylRKS : ARRAY[0..24] OF BOOL; (* Cylinder in Limp Home RKS Mode *)
	bLimpHomeCyl : ARRAY[0..24] OF BOOL; (* Cylinder in Limp Home *) (* OldName: bLimpHomeCyl; Cycle: 2 *)
	bLimpHomeAll : ARRAY[0..24] OF BOOL; (* Cylinder in any limp home mode *)
	bLimpHomeAny : BOOL; (* Any cylinder in any limp home mode *)
	bFreezeOptiCyl : ARRAY[0..24] OF BOOL; (* Cylinder Optimizer freezed *) (* OldName: bFreezeOptiCyl; Cycle: 2 *)
	bLimpHomeCylTrip : ARRAY[0..24] OF BOOL; (* Cylinder Trip because Limp Home *) (* OldName: bLimpHomeCylTrip; Cycle: 2 *)
	bHiCtr_SkipCyl : ARRAY[0..24] OF BOOL; (* Skip Cylinder HiCtr *) (* OldName: bHiContrCyl_SkipCyl; Cycle: 2 *)
	bHiCtr_IP_Ena : BOOL; (* Enable HiContr Ignition Point Offset *) (* OldName: bZZP_HierarchyCont; Cycle: 2 *)
	rCA_HiCtr_IP_Offs : REAL; (* Ignition Point Offset High controller *) (* OldName: ssHiGlobEng_ITGlobOffsetPmax; Cycle: 2 *)
	bHiCtr_MFCtr_Ena : BOOL; (* High control Misfire control enable *) (* OldName: bHiContrCyl_MFContrEnable; Cycle: 2 *)
	bTripCyl : ARRAY[0..24] OF BOOL; (* Cylinder Trip Information *) (* OldName: newPV; Cycle: 2 *)
	rHiCtr_Misf_Int : ARRAY[0..24] OF REAL; (* High Controller Misfire integrator *)
	rPI_Dur_CppInt_Offset : ARRAY[0..24] OF REAL; (* CPP Integrator Port Injection Duration reduction offset [%] *)
	rCA_Ign_CppInt_Offset : ARRAY[0..24] OF REAL; (* CPP Integrator Ignition Point reduction offset [°CA] *)
	xTOF_CppInt_P_Red : TOF; (* Off delay Nominal Power slope for Power reduction by CPP Integrator *)
	bCppInt_SkipCyl : ARRAY[0..24] OF BOOL; (* Cylinder Peak Pressure Integrator Skip Cylinder Ignition on Engine Shutdown *)
	bCppInt_OptFreeze : ARRAY[0..24] OF BOOL; (* Cylinder Peak Pressure Integrator Freeze Optimizer *)
END_VAR
(* skip_zde *)
VAR
	TOF_Skip : ARRAY[0..24] OF TOF; (*Baustein für das verzögerte Akzeptieren von Misfire Erkennungen der SAFI nach dem Skippen*) (* Statistic *)
	bIdx_Eng_SkipF : BOOL; (* Engine is Skipping *)
	iNum_SkipCyl_Act : INT; (* actual amount of skipping cylinder *) (* OldName: ssHiGlobEng_visSkipCylNr; Cycle: 2 *)
	iNum_SkipCyl_Vis : INT; (* actual amount of skipping cylinder for VISU*)
	iNum_SkipCyl_Calc : USINT; (* calculated amount of skipping cylinder *) (* Oldname: ucFixMisfPos; Cycle: 2*)
	bSkipCylAct : ARRAY[0..24] OF BOOL;
	iMisfCyl_SF : UDINT;
	bSkip_Idle : BOOL; (* Engine is in Idle and skipping *) (* Oldname: bskippen_IT; Cycle: 2*)
END_VAR
(* GEN2 *)
VAR
	bGen2_LeanoxDev_Dis : BOOL; (* Deactivate Leanox deviation error (A1080) *) (* Oldname: bLeanoxAbwAUS_GENII; Cycle: *)
	rPr_Leanox_Set_Gen2 : REAL; (* Gen2 Leanox pressure setpoint *) (* Oldname: p2s_cmd_leanox/100; Cycle: *)
	rLam_Gen2 : REAL; (* Lambda from Gen2 Controller *)
	iSkip_Gen2 : INT; (* Gen2 Skip Cylinder amount*) (* Oldname: MCL_N_skip; Cycle: *)
	bGEN2_EG_Lim_ON : BOOL := TRUE; (* SimSo_Texh_LIMIT_ON *) (* Oldname: SimSo_Texh_LIMIT_ON; Cycle: *)
	LCRRamp_Lambda_Gen2 : LCRRamp;
END_VAR
(* PBC *)
VAR
	bIPC_MSF : ARRAY[0..24] OF BOOL; (* in-cylinder pressure sensor measuring signal failure *) (* OldName: bDMRFault,bFadOutCyl_SensF; Cycle:2; *)
	tWarn_IPC_MSF : AmmSequence; (* Warn: A2577, OM: B2802, Cylinder pressure sensor measuring signal failure *) (* OldName: bWDMRSigErr, bBDMRSigErr, ucDMRSigErr; Cycle: 2 *)
	rPr_CPP_Min : REAL;
	rPr_CPP_Max : REAL;
	rPr_IMEP_Min : REAL;
	rPr_IMEP_Max : REAL;
	rCA_MFBvar_Min : REAL;
	rCA_MFBvar_Max : REAL;
	rPr_CPP_Avg : REAL;
	rPr_IMEP_Avg : REAL;
	rCA_MFBvar_Avg : REAL;
	rPr_49bfTDC_Min : REAL;
	rPr_49bfTDC_Max : REAL;
	rPr_49bfTDC_Avg : REAL;
	rPr_Knck_Min : REAL;
	rPr_Knck_Max : REAL;
	rPr_Knck_Avg : REAL;
END_VAR
(* pv_check *)
VAR
	tOM_EngineMap : AmmSequence; (*OM: B2826, Engine map automatically loaded*) (* OldName: bAPmaxAbsLimit, bBPmaxAbsLimit, ucPmaxAbsLimit; Cycle: 2 *)
END_VAR
(* wastegate *)
VAR
	bErr_WG_MSF : BOOL := FALSE;
	bErr_WG_MSF_A : BOOL := FALSE;
	bErr_WG_MSF_B : BOOL := FALSE;
	bErr_WG_Dev : BOOL := FALSE;
	bErr_WG_Dev_A : BOOL := FALSE;
	bErr_WG_Dev_B : BOOL := FALSE;
	bWG_Check : BOOL := FALSE;
END_VAR
(* TC1 SPP *)
VAR
	rPr_GR_TC1 : REAL; (* GR Filt TC1*)
	rPr_P1_TC1 : tBank_AB; (* P1 Filt TC1*)
	rPr_P2s_TC1 : tBank_AB; (* P2s Filt TC1*)
	rPr_EGaHP_TC1 : tBank_AB; (* P3s Filt TC1*)
	rPr_EGaLP_TC1 : tBank_AB; (* P4 Filt TC1*)
END_VAR
(* FastStart *)
VAR
	rCA_IP_StartOffs : REAL; (*ignition point start offset*)
	rCA_IP_EGTCtr_Offs : REAL; (*ignition point EGTCtr offset*)
	rCA_IP_StartOffs_speed : REAL; (*ignition point start offset speed ramp*)
	rP_LR_Trig_ActSat_TV : REAL;
	rTi_LR_ActSat_TV : REAL;
	rN_LR_CBV_SAT_ON : REAL;
	rP_LR_Trig_GasStop : REAL;
	rP_LR_GCB_Trig_GasStop : REAL; (*Trigger value of load rejection at opening of GCB to close gas valve (Tejcet) and set actuators (open CBP, close TV) [%]*)
	rP_LR_GCB_Trig_Misf : REAL; (*Trigger value of load rejection at opening of GCB to activate misfire function[%]*)
	rLR_Gasstop_CBV_Man : REAL;
	rTi_LR_GasStop_OFF : REAL;
	rTi_LR_GasStop : REAL;
	rP_LR_Trig_Misf : REAL;
	rN_Misf_2_Trig : REAL;
	iCycles_MisfireActive : INT; (*Parameter: number of engine cycles the misfire function should be active *)
	rTi_LR_IGN_Retard_MAX : REAL;
	rP_LR_Trig_IGN_Retard : REAL;
	rN_LR_IGN_Retard_ON : REAL;
	rN_TV_Release_Lim_Max : REAL;
	rN_TV_Release_Lim_Min : REAL;
	rPosTV_CBV_Release_Max : REAL;
	rN_trig_cbv_lim : REAL;
	iTime_Cyc : INT := 0;
	iTime_Eng_Cyc : INT := 0;
	iCyc_Ign_Max_Off : INT := 0;
	iCyc_Ign_Min_On : INT := 0;
	tLock_TV_PT : TIME;
	rLockTV_Rise : REAL;
	rLockTV_Sink : REAL;
	rP_Trig_TVbyP2S_OFF : REAL;
	tLIM_TVbyP2s_OFF_PT : TIME;
	rN_LIM_TVbyPOS_ON : REAL;
	bLIMIT_TVbyP2s_act : BOOL;
	bLIMIT_TVbyCBV_act : BOOL;
	xTOF_LIM_TVbyP2s_OFF : TOF;
	bLIM_TVbyP2s_OFFatLargeRej : BOOL;
	bLIM_CBV_by_TVpos : BOOL;
	bUseKPduringSaturation : BOOL;
	rTi_LR_Overwrite_CBV : REAL;
	rN_LR_Overwrite_CBV_START : REAL;
	rN_LR_Overwrite_CBV_END : REAL;
	bInitCBV_const : BOOL;
	bLR_CBV_Overwrite : BOOL;
	bLR_CBV_Overwrite_Act : BOOL;
	rLR_CBV_Overwrite_Init : REAL;
	rLR_CBV_Overw_InitOffset : REAL;
	iT_filt_INPUT_u_cbv : UINT;
	rP_LR_Trig_Overwrite_CBV : REAL;
	rN_LR_CBV_GainMult : REAL;
	rLR_CBV_GainMult_high : REAL;
	rLR_CBV_GainMult_low : REAL;
	rLamAdapt_Ramp_Grad : REAL;
	rLamAdapt_Ramp_Grad_LowSpeed : REAL;
	rN_LamAdapt_Ramp_Switch : REAL;
	rP_LamCorrAct_Max_Norm : REAL;
	Kp_CBV_LR_Overwrite_data : ARRAY[0..4] OF lcrCurveByPoints_TabEntry_type;
	tMisfprotect_OFF_PT : TIME;
	rN_CBV_Release_Lim_Min : REAL;
	rP_LamSlowLamRamp : REAL;
	bFiltInputVolFlow_TEST : BOOL;
	rP_Rot_Norm_Lam_Save_Trig : REAL;
	xLCRCurve_Dyn_Lambda_LimD_table : ARRAY[0..4] OF lcrCurveByPoints_TabEntry_type;
	rP0_Nom : REAL;
	rP_Ramp_FC_max_Gen1 : REAL;
	rP_Ramp_FC_max_Gen2 : REAL;
END_VAR
```

### Program Logical/EngineController/IN_EngCtr (IEC, version 4.14.0) - + Engine Controller input task

- IN_EngCtr.st (not readable text: treated as protected, skipped)

#### IN_EngCtr.var - Local variables
```iecst
(********************************************************************
 * COPYRIGHT -- INNIO Company
 ********************************************************************
 * Program: IN_EngCtr
 * File: IN_EngCtr.var
 * Author: 502293141
 * Created: March 03, 2015
 ********************************************************************
 * Local variables of program IN_EngCtr
 ********************************************************************)
VAR
	ti_Cycle_lim : TIME;
	ti_Cycle : TIME;
	xSS : SS;
	xSS_WG : SS_Cust := (0);
	xSS_PFPDR : SS_Cust := (0);
	xSS_Opt : SS_Cust := (0);
	xSS_LamLim : SS_Cust := (0);
END_VAR
VAR CONSTANT
	_SS_P2s : USINT := 1;
	_SS_T2s : USINT := 2;
	_SS_T_EG : USINT := 4;
	_SS_P_Norm : USINT := 8;
	_SS_Pd_Norm : USINT := 64;
END_VAR
VAR
	xTON_Amb : TON;
	xFILTER_Pr_Amb : FILTER_R;
	iMainMode_OP : INT := 0;
	iMainMode_OP_Last : INT := 0; (* operation mode from the previous cycle *)
	iMainMode_OP_Prev : INT := 0; (* operation mode from the previous operation *)
	rN_limit_norm_Gen2Idle : REAL := 0.005; (*if GCB OFF and speed in tolerance band around Nnom switch to Idle controller*)
	bDeactIdleAfterGCBoff : BOOL := FALSE; (* Only island controller active after GCB off *)
	bSpeed_recovered_afterGCBoff : BOOL := FALSE; (* speed inside tolerance band after GCB off*)
	bRelease_IdleCtr_afterGCBoff : BOOL := FALSE; (*Idle controller released after GCB off*)
	bForce_Gen2island_afterGCBoff : BOOL := FALSE;
	TP_force_Gen2island_afterGCBoff : TP;
	rT_force_Gen2island_afterGCBoff : REAL := 1.0; (* [s] time to force Gen2 island after GCB off *)
	TP_wait_SpeedRecovered : TP;
	rTWait_Release : REAL := 5.0; (* [s] time to delay the release for idle control after speed recovered *)
	bSpeed_recovered_delay : BOOL := FALSE; (* speed inside tolerance band after GCB off and waiting time TWait_Release over*)
	rP_Act_Norm_GCBoff : REAL := 0.0; (* normalized power at time when GCBoff *)
	rPmin_norm_Gen2idle : REAL := 0.2; (* normalized minimal power at time GCBoff to activate Gen2*)
	LCRCurveByPoints_VE_Eng_P2s : LCRCurveByPoints; (* linear interpolation function for volumetric efficiency boost pressure dependency *)
	LCRCurveByPoints_VE_Eng_T2s : LCRCurveByPoints; (* linear interpolation function for volumetric efficiency charge temperature dependency *)
	LCRCurveByPoints_VE_Eng_N : LCRCurveByPoints; (* linear interpolation function for volumetric efficiency speed dependency *)
	rVE_Eng_P2s : REAL; (* volumetric efficiency boost pressure dependency *)
	rVE_Eng_T2s : REAL; (* volumetric efficiency charge temperature dependency *)
	rVE_Eng_N : REAL; (* volumetric efficiency speed dependency *)
	xTOF_SyDemand : TOF; (* Grid Status Detection: TOF block for function reset after SY *)
	tiOf_afterIdle : TIME := T#5s; (* Grid Status Detection: TOF time for function reset after SY*)
	bResetGridStat : BOOL; (* Grid Status Detection: manual reset of function *)
	xTP_GCB_DCon : TP;
	bTrig_GCB_DCon_EC : BOOL;
	tiTrig_Duration : TIME := T#2s;
	xTON_ParaOK_Lp_c_Ena : TON;
	bGEN2island_T6premixed : BOOL := FALSE; (* Release GEN2 island for T6 premixed *)
	LCRCByP_rEtaVolOffs : LCRCurveByPoints; (* T4 vol. efficiency offset depending on p2s*)
	refPoint_rEtaVolOffs : ARRAY[0..5] OF lcrCurveByPoints_TabEntry_type;
	rQ_offset : REAL; (* offset to shift reactive power range to posite range 0-Qnom [kVAr] *)
	rQ_nom : REAL;  (* reactve power range [kVAr] *)
END_VAR
```

### Program Logical/EngineController/gen_EC_T2 (IEC) - + common tasks @ 10ms

- gen_EC_T2.st (not readable text: treated as protected, skipped)

#### gen_EC_T2.var - Local variables
```iecst
(********************************************************************
 * COPYRIGHT -- INNIO Company
 ********************************************************************
 * Program: general_EC
 * File: general_EC.var
 * Author: WaldharM
 * Created: May 22, 2012
 ********************************************************************
 * Local variables of program general_EC
 ********************************************************************)
VAR
	TOF_Act_Release : TOF;
	TON_Act_Mon_Release : TON;
	TON_WGActDO : TON;
	TON_Act_Mon_Rel_WG : TON;
	bWG_Dem_Active : BOOL := 0; (* general wastegate demand *)
	iConf_WG_EEPROM : INT := 0; (*EEPROM configuration state*)
	tDataSend_WG_EEPROM : ARRAY[0..7] OF BYTE := [8(0)]; (*WG data to send to EEPROM*)
	tDataSend_WG_ID : ARRAY[0..7] OF BYTE := [8(0)]; (*WG data to send to EEPROM*)
	bEEPROMRead : BOOL := 0; (*Config EEPROM read modus*)
	bEEPROMWrite : BOOL := 0; (*Config EEPROM write modus*)
	iConf_WG_EEPROM_Next : INT := 0; (*next EEPROM configuration step*)
	xTON_WG_EEPROMTransfer : TON := (0); (*Timer to EEPROM Transfer*)
	bTON_WG_EEPROMTransfer : BOOL := 0; (*Trigger timer to EEPROM Transfer*)
	xTON_WG_EEPROMReading : TON := (0);(*Timer to EEPROM Reading*)
	bTON_WG_EEPROMReading : BOOL := 0; (*Trigger timer to EEPROM Reading*)
	xTP_WG_EEPROMReadLim : TP := (0); (*Timer EEPROM Read Actuator Info*)
	xTON_WG_ConfigReset : TON := (0); (*Timer to reset CAN WG actuators*)
	xTON_WG_WaitingConfig : TON := (0); (*Timer to stop configuration if actuator not responsding*)
	bTON_WG_Conf_Reset : BOOL := 0; (*Trigger timer to reset CAN WG actuators set flag*)
	bTON_WG_WaitConfig : BOOL := 0; (*Trigger timer to stop configuration if actuator not responsding*)
	tCAN_WG_ReqSN : ARRAY[0..3] OF BYTE := [4(0)]; (*CAN wastegate request serial number addresses*)
	tCAN_WG_ReqSw : ARRAY[0..3] OF BYTE := [4(0)]; (*CAN wastegate request software version addresses*)
	tCAN_WG_ReqOpH : ARRAY[0..1] OF BYTE := [2(0)]; (*CAN wastegate request operating time addresses*)
	tCAN_WG_ReqSrcAdd : ARRAY[0..1] OF BYTE := [2(0)]; (*CAN wastegate request source address addresses*)
	sWG_CAN_Sw_Tmp : STRING[12] := '000000000000'; (*CAN WG actuator software version - TEMPORARY variable*)
	sWG_CAN_SN_Tmp : STRING[10] := '0000000000'; (*CAN WG actuator serial number - TEMPORARY variable*)
	tWG_CAN_OpH_Tmp : ARRAY[0..3] OF BYTE := [4(0)]; (*CAN WG actuator operating time [h] - TEMPORARY variable*)
	tWG_CAN_ActSrcAdd_Tmp : BYTE := 0; (*CAN WG actuator source address - TEMPORARY variable*)
	iReq_WG_Data : USINT := 0; (*CAN wastegate request data - MSG indexing*)
	tWG_CAN_EEPROM_Msg : BYTE := 0; (*CAN wastegate expected MSG (0-7 BITS) general*)
	tWG_CAN_A_EEPROM_Msg : BYTE := 0; (*CAN wastegate expected MSG (0-7 BITS) WG_A*)
	sTmp_WG_CAN : STRING[4] := ''; (*Temp variable CAN read message*)
	tWG_CAN_B_EEPROM_Msg : BYTE := 0; (*CAN wastegate expected MSG (0-7 BITS) WG_B*)
	bWG_CAN_A_ReadEEPROM : BOOL := 0; (*Info (S/N,Sw Vers,OpH,SrcAdd) Device A Read Modus*)
	bWG_CAN_B_ReadEEPROM : BOOL := 0; (*Info (S/N,Sw Vers,OpH,SrcAdd) Device B Read Modus*)
	bWG_ReadFunction : BOOL := 0; (*read device Info can be done *)
	iCnt_OpHours_Old : DINT := 0; (*actual OpH*)
	bWG_CAN_A_OpH_Reading : BOOL := 0; (*OpH Device A Read Modus*)
	bWG_CAN_B_OpH_Reading : BOOL := 0; (*OpH Device B Read Modus*)
	bWG_CAN_A_Reading : BOOL := 0; (*Info WG_A Reading*)
	bWG_CAN_B_Reading : BOOL := 0; (*Info WG_B Reading*)
	bWG_CAN_A_Learn_On : BOOL := 0; (*WG CAN A Learn State*)
	bWG_CAN_B_Learn_On : BOOL := 0; (*WG CAN B Learn State*)
	bCAN_WG_Dem_Active : BOOL := 0; (*CAN Wastegate demand active*)
	bWG_CAN_OpH_Rdy : BOOL := 0; (*Reading OpH Ready*)
END_VAR
```

- Logical/EngineController/eng_ctr_EC (protected, skipped)

### Program Logical/EngineController/Gen2_xt (IEC) - + GEN2 controller

- Gen2_xtCyclic.st (not readable text: treated as protected, skipped)

- Gen2_xtInit.st (not readable text: treated as protected, skipped)

#### Gen2_xt.var - Local variables
```iecst
(********************************************************************
 * COPYRIGHT -- INNIO Company
 ********************************************************************
 * Program: Gen2_xt
 * File: Gen2_xt.var
 * Author: 502427335
 * Created: June 18, 2015
 ********************************************************************
 * Local variables of program Gen2_xt
 ********************************************************************)
VAR
	roffset_Ug : REAL; (*offset generator voltage*)
	bFreqM_Gen2 : BOOL; (*Insel: Motordrehzahl wird über Generatorfrequenz berechnet*)
	LCRCByP_LamLoLim_ABS : LCRCurveByPoints;
	TON_LOXErr : TON;
	bResetGlobal_Man : BOOL;
	LCRCByP_SkipFkp : LCRCurveByPoints;
	LCRCByP_SkipFLevel : LCRCurveByPoints; (* overspeed threshold to start skip fire with respect to power  *)
	LCRCByP_PwrCtrKi : LCRCurveByPoints;
	LCRCByP_rEtaBrakeExt : LCRCurveByPoints;
	LCRCByP_rGain_iLQR_rR0 : LCRCurveByPoints;
	p2_offset : REAL;
	sstrace : INT := 2;
	TON_LeanoxDev_Dis : TON;
	TON_Trigger : TON;
	tAbtastT : TIME := T#5s;
	rMAX : REAL;
	rMIN : REAL;
	rP_Leanox_bloc : REAL := 0.01;
	rGen2_rP_Set_old : REAL;
	rGen2_rP_des_old : REAL;
	rP_LimitBDC_Norm : REAL;
	TON_Pelmax : TON;
	rP0_Nom_normal : REAL;
	rhoAir : REAL := 1.293;
	bSaveLamOffsetLim : BOOL := 0;
	nc : INT := 0;
	bGEN2_calconly : BOOL := FALSE;
	bActGasMixGen2 : BOOL := TRUE;
	TON_SaveLam : TON;
	bReleaseAutoLamSave : BOOL := TRUE;
	bInitTvActPos : BOOL := TRUE;
	bInitLamMin : BOOL := TRUE;
	tLamSaveTime : TIME := T#5m;
	bIsland_old : BOOL;
	p2s_offset : REAL;
	Pel_offset : REAL;
	rP_Ramp_Dec_Fast : REAL := 0.1;
	bSaveKeMap : BOOL := FALSE;
	rMinKpSkip : REAL := 0.0;
	rTiFpowtraj : REAL;
	bGS_TBDC : BOOL := FALSE;
	LCRCByP_TBDC : LCRCurveByPoints;
	refPoint_TBDC : ARRAY[0..5] OF lcrCurveByPoints_TabEntry_type;
	rTiBDC_OvSpd : REAL;
	rN_TBDC_OvSpd : REAL;
	rR0_OvSped : REAL;
	rR0 : REAL;
	bR0_OvSped : BOOL;
	bTiBDC_OvSpd : BOOL;
	rP_Diff_Max_Norm_old : LREAL;
	minPawLam : REAL;
	Para_rGEN2_ResetKe_z : REAL := 0.0;
	rK_LEANOX : REAL := 0.0;
	rKd_skiplevel : REAL := 0.0;
	bReset_Ke : BOOL := FALSE;
	rP0_Nom_normal_type6 : REAL;
	rPr_p2s_Idle : REAL; (*[bar] latest p2s in idle operation*)
	bIdle_old : BOOL;
	rPr_desired_p2s_min : LREAL; (*[bar]*)
	rPr_lowLoad_p2s_min : REAL; (*[bar]*)
	TON_NetP : TON;
	xRAMPE_p2s_0kW : RAMPE_R;
	rT_EO_Idle : REAL; (*[degC] latest TOil in idle operation*)
	rStd_Ramp_p2s_0kW : REAL;
	rT_EO_Nom : REAL := 70; (*[degC] reference engine oil temperature above which the engine will be classified as hot*)
	bBlock_LamAdaptSY : BOOL;
	rLam_min_adapt : REAL;
	rFact_LamAdapt : REAL;
	rLam_Idle : REAL; (*[-] latest lambda in idle operation*)
	rLam_min_atIdle : REAL;
	rLam_initialOffset : REAL := 0.2; (*[pu] amount of delta in lambda which will be released immediatly after SY*)
	TON_NetPLONG : TON;
	bBlock_p2s_0kW_AdaptSY : BOOL; (*TRUE = starr/ramp up phase is done and the SY/low load adaption is blocked*)
	TON_NetP20s : TON;
	rFacRampDown_lowLoad : REAL := 1.4; (*factor for p2s_set for low load in hot engine condition*)
	rFacRampDown : REAL := 1.2; (*factor for p2s_set for low load dunring ramp down*)
	rP2s_0kW_optimal_T6_TSTC : REAL := 0.40; (*[bar] base p2s set value for type 624*)
	rP2s_0kW_optimal_T6_SSTC : REAL := 0.36; (*[bar] base p2s set value for type 612/616/620*)
	rP2s_0kW_optimal_T34 : REAL := 0.3; (*[bar] base p2s set value for type 3 and 4*)
	rIP_Pset : REAL;
	rIP_Pset_min : REAL := 0.125; (*[pu] min. Power below that the maximum p2s_set increasing will be used for engine ramp down or low load after the start function is blocked*)
	rIP_Pset_max : REAL := 0.2; (*[pu] max. Power above that no p2s_set increasing will be used for engine ramp down or low load after the start function is blocked*)
	tDelNetpMLong : TIME := T#15m; (*max. Time after GCB_on the p2s_set adatpion for T6 is activated*)
	bGEN2_T6_LowLoadImpr_Active : BOOL := TRUE; (*TRUE = GEN2 Low Load imrovement activated*)
	refPoint_ff2load_lim_fact : ARRAY[0..3] OF lcrCurveByPoints_TabEntry_type;
	LCRCByP_ff2load_lim_fact : LCRCurveByPoints;
	rLSLff2load_lim_fact : REAL := 1.0;
	bNetP_z : BOOL;
	bSaveKeMap_transition : BOOL;
	rTiF_KeEstDiffMapUpdate : REAL := 10.0; (* [s] Filter time const. for Ke_est - Ke_map to update Keng Map*)
	rLam_Start_init : REAL := 0.000; (*init value PowCtrl.rLam_Start *)
	rFactGQCP2sOffsMax : REAL := 0.2;
	bEnableFuncQGC : BOOL := TRUE; (*enable functions for gas qual. Changes: p2s offset, lambda external*)
	rN_Gen2_InMixSpdFreq_fact : REAL := 0.0; (*Factor for mixing of speed and frequency signals for Load Rejection Calculations*)
	rN_Gen2_InMixSpdFreq_norm : REAL := 1.0; (*Normalized frequency used for calculated speed trigerring load rejections*)
	rNskip_Gen2FactorMax : REAL := 1.0; (* GEN2 factor maximal number of skipped cylinders *)
	iNskip_Gen2Max : INT; (* GEN2 maximal number of skipped cylinders *)
	iNskip_Gen2 : INT; (* GEN2 number of skipped cylinders *)
	rT_EG_COLD : REAL := 100;
	xTON_GCB : TON;
	bEngineHot : BOOL; (*TRUE = Engine in hot condition*)
	rGain_speed2boost_iLQR : REAL := 0.1;
	rGain_ss_speed_iLQR_back_cold : REAL := 1.0;
	rGain_ss_speed_iLQR_back : REAL := 0.15;
	rGain_ss_boost_iLQR_cold : REAL := 0.001;
	rT_EG_HOT : REAL := 500;
	refPoint_SkipFkp : ARRAY[0..1] OF lcrCurveByPoints_TabEntry_type;
	rTcMaxSpeed_Buffer : REAL;
	bActive_UnitTestFRTisland : BOOL;
	bFlag_GEN2FRTisland : BOOL;
	ti_TOFGEN2FRTisland : TIME := T#10ms;
	xTOF_GEN2FRTisland : TOF;
	rGen2_LoadEstNu : REAL := 2.0000;
	rGen2_LoadEstNu_FRT : REAL := 0.0000;
	bFRT_GEN2active : BOOL := TRUE; (*Activation GEN2 reaction on FRT island detection*)
	rP_Th_LR_DBOV : REAL; (* rotational power threshold for DBOV activation at load rejections *)
	rN_Th_LR_DBOV_norm : REAL; (* normed speed threshold for high PI CUrrent activation at load rejections *)
	xTP_LR_DBOV : TP; (* time pulse for DBOV activation at load rejections *)
	rP_GEN2_T6LoLoadLearning_Lim : REAL := 0.1; (* GEN2 island T6PreM *)
	xGR_MINR_GEN2T6LoLoadLearn : GR_MINR; (* GEN2 island T6PreM *)
	rLam_EOT_GEN2offs : REAL := 0.2; (* GEN2 island T6PreM *)
	rR_iLQR_0_LowLoad : REAL := 20; (* GEN2 island T6PreM *)
	rR_iLQR_1_LowLoad : REAL := 1000000000; (* GEN2 island T6PreM *)
	rQ_iLQR_1_LowLoad : REAL := 0.0; (* GEN2 island T6PreM *)
	rQ_iLQR_2_LowLoad : REAL := 0.0; (* GEN2 island T6PreM *)
	rQ_iLQR_1_LowLoad_wKF : REAL := 0; (* GEN2 island T6PreM *)
	rQ_iLQR_0_LowLoad_wKF : REAL := 1.0; (* GEN2 island T6PreM *)
	ti_GEN2_p2sManActiveTOF : TIME := T#10s;
	xTOF_GEN2_p2sManActive : TOF;
	bLP_c_Ena_Gen2 : BOOL; (*enable Leanox point C for Gen2*)
	refPoint_rITPoffsetP2s : ARRAY[0..4] OF lcrCurveByPoints_TabEntry_type; (* Gen2 IT Offset in NetP *)
	LCRCByP_ITPoffsetP2s : LCRCurveByPoints;
	xRAMPE_LamLim_BackfPrev : RAMPE_R;
	rFactEnrich_BackfPrev : REAL := 0.7; (*Enrichment amplitude scaling for combustion anomaly detection*)
	rK_FSM_WO_0 : REAL := 0.0;
	rDp_Gasrail_max : REAL; (* Maximum differential pressure across PI-Valve *)
	T_TripLnxOff : TIME := T#280s;
	rGainLamUplim2boost : REAL := 0.0;
	rGainLamUplim2boostOvSpd : REAL := 0.0;
END_VAR
```

### Program Logical/EngineController/WasteGate (IEC) - + interface for WG outputs

- WasteGate.st (not readable text: treated as protected, skipped)

#### WasteGate.var - Local variables
```iecst
(********************************************************************
 * COPYRIGHT -- INNIO Company
 ********************************************************************
 * Program: WasteGate
 * File: WasteGate.var
 * Author: 105051472
 * Created: November 22, 2010
 ********************************************************************
 * Local variables of program WasteGate
 ********************************************************************)
VAR
	xRAMPE_WasteGate : RAMPE_R; (*FUB*)
	xTON_Dev : TON;
	xTON_Dev_A : TON;
	xTON_Dev_B : TON;
	rPos_WG_DevMax : REAL := 0.05;
	xTON_WG_Act : TON;
	xTON_WG_Act_A : TON;
	xTON_WG_Act_B : TON;
	xTON_bErrMsWasteGate : TON;
	xTON_bErrMsWasteGate_A : TON;
	xTON_bErrMsWasteGate_B : TON;
	xLCRPT1_CBV : LCRPT1;
	rTConst_CBV : REAL;
	bELR : BOOL := 0;
	bHys_Inc_WG : BOOL := 0;
	bHys_Dec_WG : BOOL := 0;
	xTON_ELR : TON;
	iWG_State : USINT;
	bWG_Check_Rel : BOOL;
	xTON_WG_Wait : TON;
	xTON_WG_Open : TON;
	xTON_WG_Close : TON;
	xRS_Transient : RS;
	bWG_Ctrl_ON : BOOL; (*Wastegate controller active*)
	xR_TRIG_bFreeze_GEN2 : R_TRIG; (* trigger activation of GEN2 freeze to keeep CBV tracking on  *)
	xR_TRIG_bSS_GEN2 : R_TRIG; (* trigger activation of steady state to keeep CBV tracking on  *)
	bForceGen2CBVtracking : BOOL; (* force CBV tracking bit after grid event *)
	bGEN2_Ctrl_WG_NP : BOOL; (* WG control by GEN2 enabled for net parallel *)
	bGEN2_Ctrl_WG_Island : BOOL; (* WG control by GEN2 enabled for isolated operation *)
END_VAR
VAR CONSTANT
	OPEN : USINT := 3;
	WAIT : USINT := 1;
	CLOSE : USINT := 4;
	INACT : USINT := 0;
	ACT : USINT := 2;
END_VAR
VAR
	tDataRec_WG_A : ARRAY[0..7] OF BYTE := [8(0)]; (*WG A CAN read actuator status*)
	tDataRec_WG_B : ARRAY[0..7] OF BYTE := [8(0)]; (*WG B CAN read actuator status*)
	tDataRec_Err_WG_A : ARRAY[0..7] OF BYTE := [8(0)]; (*WG A CAN read actuator faults and warnings*)
	tDataRec_Err_WG_B : ARRAY[0..7] OF BYTE := [8(0)]; (*WG B CAN read actuator faults and warnings*)
	iT_Tmp : INT := 0; (*WG CAN internal temperature*)
	iWG_ReadActWarn : USINT := 0; (*WG CAN actuator warning ID in status*)
	iWG_ReadActFail : USINT := 0; (*WG CAN actuator failure ID in status*)
	bWG_CAN_A_Fail : BOOL := 0; (*WG A CAN Failure trigger bit*)
	bWG_CAN_A_Warn : BOOL := 0; (*WG A CAN Warning trigger bit*)
	bWG_CAN_B_Fail : BOOL := 0; (*WG B CAN Failure trigger bit*)
	bWG_CAN_B_Warn : BOOL := 0; (*WG B CAN Warning trigger bit*)
	bCANread_WG_A_St : BOOL := 0; (*WG A CAN read status*)
	bCANread_WG_B_St : BOOL := 0; (*WG B CAN read status*)
	bTON_CANcomm_WG_A_Err : BOOL; (*WG A CAN communication error trigger bit*)
	bTON_CANcomm_WG_B_Err : BOOL := 0; (*WG B CAN communication error trigger bit*)
	xTON_CANcomm_WG_A_Err : TON := (0);
	xTON_CANcomm_WG_B_Err : TON := (0);
	xTON_CAN_WG_A_FailWarn : TON := (0);
	xTON_CAN_WG_B_FailWarn : TON := (0);
	xTON_WG_A_CANcomm : TON := (0);
	xTON_WG_B_CANcomm : TON := (0);
	iT_WG_Offset : UINT := 0;
	bErr_WG_CANcomm : BOOL := 0;
END_VAR
```

### Program Logical/EngineController/gas_flow_EC (IEC) - + calculation gasflow for gas inject valve

- gas_flowCyclic.st (not readable text: treated as protected, skipped)

- gas_flowInit.st (not readable text: treated as protected, skipped)

#### gas_flow.var
```iecst
VAR
	a : ARRAY[0..3] OF REAL;
	af : ARRAY[0..3] OF REAL;
	AmmSeqGASM : AmmSequence;
	AmmSeqGASO : AmmSequence;
	an : ARRAY[0..3] OF REAL;
	an_f : ARRAY[0..3] OF REAL;
	b : ARRAY[0..3] OF REAL;
	bAdmitCtrl : BOOL;
	bAdmitFlow : BOOL; (* TRUE=gas flow is admited *)
	bf : ARRAY[0..3] OF REAL;
	bn : ARRAY[0..3] OF REAL;
	bn_f : ARRAY[0..3] OF REAL;
	bPumpErkennung : BOOL;
	bSpeedCorr : BOOL; (*Drehzahlkorrektur ist ein*)
	FILTER_R_T2s_RAW : FILTER_R;
	FILTER_R_P2_RAW : FILTER_R;
	FILTER_R_P2s_RAW : FILTER_R;
	FILTER_R_P2s_50ms : FILTER_R; (* FUB filter boost pressure T=50 ms *)
	LCRMovAvg_tg : LCRMovAvgFlt;
	rFlow_GMK_Lo : REAL;
	rFlow_GMK_Hi : REAL;
	P2s_NReg_DigFil : DigFil;
	P2s_TJ_DigFil : DigFil;
	P2_NReg_DigFil : DigFil;
	P2_TJ_DigFil : DigFil;
	RAMPE_AddGas : RAMPE;
	RAMPE_MixGas : RAMPE; (* limit gas mixture change speed *)
	rCF_TV_Ctr : REAL;
	rCF_CBV_Ctr : REAL;
	rCBV_Comp_Amt : REAL;
	rCF_Speed : REAL; (*Drehzahlkorrektur*)
	rCorr_Pr : REAL; (*Preassure Compensation*)
	rCorr_T : REAL; (*Temp correctur factor*)
	rDkScal2 : REAL;
	rCF_Rot : REAL; (* Correction factor Volumenstrom Rotation *)
	rPos_CBV_dt : REAL; (* Letzte CBV Änderung *)
	rCF_CBV_dyn : REAL;
	rCF_TV_dyn_rated : REAL;
	rCF_TV_dyn : REAL;
	rCF_TV_dyn_lim : REAL;
	rCF_CBV_dyn_lim : REAL;
	rFlow : REAL; (* Volumenstrom Engine [m3/s] *)
	rFlowDiff : REAL;
	rFlowDiffM : REAL;
	rFlowMax : REAL; (* max. allowed gas flow*)
	rFlowMaxDiff : REAL;
	rFlowMaxDiffM : REAL;
	rFlowMaxM : REAL; (* max. allowed gas flow gas train 2 *)
	rFlowScal2 : REAL;
	rFlow_reg : REAL; (* Volumenstrom Engine reg [m3/s] *)
	rCF_CBV_dt : REAL; (* compensation by relativ turbo bypass compensation *)
	rGasFlow : REAL; (*setpoint gasflow whole engine*)
	rGasFlowM : REAL; (*setpoint gasflow gas train 2*)
	rJkorr : REAL;
	rN_LamCorr : REAL := 0.0; (* value speed dependend compensation *)
	rCF_Lam_Speed : REAL;
	rCF_Lam_Hi : REAL := 0.0; (* constand speed dep. compensation *)
	rCF_Lam_Lo : REAL := 0.0; (* constant speed dep. compensation *)
	rLambda : REAL; (* engine lambda for calc. gas flow *)
	rLambdaAdaptGC : REAL;
	rLambdaAdaptGC_P : REAL;
	rLam_min : REAL;
	rLam_max : REAL;
	rPos_CBV_dt_f : REAL; (* Letzte CBV Änderung gefiltert *)
	rPos_CBV_dt_f_old : REAL; (* alter Wert: Letzte CBV Änderung gefiltert *)
	rMonGasFlow : ARRAY[0..4] OF REAL;
	rN_DigFil : DigFil;
	rN_Eng_df_1 : REAL; (*Drehzahl Digital gefiltert 1 [U/min]*)
	rN_Eng_df_2 : REAL; (*Drehzahl Digital gefiltert 2 [U/min]*)
	rN_Eng_df_2_dt : REAL; (*Differenz von Drehzahl Digital gefiltert 2 [(U/min)/s]*)
	rN_Set : REAL; (*Speed Setpoint Speed controller [U/min]*)
	rN_TJ_DigFil : DigFil;
	rPos_CBV_old : REAL;
	rPr_DkScal1 : REAL;
	rPr_FlowScal1 : REAL;
	rPr_P2_df : REAL; (*P2 Digital gefiltert in [bar]*)
	rPr_P2_df_TJ : REAL; (*P2 Digital gefiltert in [bar]*)
	rPumpGrenzwert : REAL;
	rPumpQuotient : REAL;
	rCF_Flow_LimLo : REAL; (* Correction Factor Limit Low *)
	rCF_Flow_LimHi : REAL; (* Correction Factor Limit High *)
	rT_GMK : REAL; (* Durchschnittliche Temperatur GMK [°C] *)
	rT_T2s_f : REAL; (* Temperatur T2s gefiltert [°C] *)
	rCF_VR_GMK : REAL; (* Correction Factor Volumenänderung in V-Raum und GMK *)
	rFlow_LIVC : REAL; (*Volumenstrom für Inselbetrieb (LIVC Regler)*)
	rFlow_CBV_dyn : REAL; (* dynamic Volumenstrom für CBV Betrieb [m3/s] *)
	rFlow_CBV_dyn_lim : REAL; (* dynamic Volumenstrom für CBV Betrieb [m3/s] *)
	rFlow_TV_dyn : REAL; (* dynamic Volumenstrom limitiert für TV Betrieb [m3/s] *)
	rFlow_TV_dyn_lim : REAL; (* dynamic Volumenstrom limitiert für TV Betrieb [m3/s] *)
	rVol_GMK : REAL; (* Volumen GMK [m3]*)
	rVol_GMK_old : REAL; (* alter Wert: Volumen GMK [m3]*)
	rVol_GMK_TJ_old : REAL; (* alter Wert: Volumen GMK (TJ filter) [m3]*)
	rVol_GMK_TJ : REAL; (* Volumen GMK (TJ filter) [m3]*)
	rVol_GMK_208 : REAL; (*208 GMK Volumen in [m3]*)
	rVol_GMK_312 : REAL; (*312 GMK Volumen in [m3]*)
	rVol_GMK_316 : REAL; (*316 GMK Volumen in [m3]*)
	rVol_GMK_320 : REAL; (*320 GMK Volumen in [m3]*)
	rVol_GMK_412 : REAL; (*412 GMK Volumen in [m3]*)
	rVol_GMK_416 : REAL; (*416 GMK Volumen in [m3]*)
	rVol_GMK_420 : REAL; (*420 GMK Volumen in [m3]*)
	rVol_GMK_424 : REAL; (*424 GMK Volumen in [m3]*)
	rVol_GMK_612 : REAL; (*612 GMK Volumen in [m3]*)
	rVol_GMK_616 : REAL; (*616 GMK Volumen in [m3]*)
	rVol_GMK_620 : REAL; (*620 GMK Volumen in [m3]*)
	rVol_GMK_624 : REAL; (*624 GMK Volumen in [m3]*)
	rVol_VR : REAL; (* Volumen VR [m3]*)
	rVol_VR_old : REAL; (* alter Wert: Volumen VR [m3]*)
	rVol_VR_TJ_old : REAL; (* alter Wert: Volumen VR (TJ filter) [m3]*)
	rVol_VR_TJ : REAL; (* Volumen VR (TJ filter) [m3]*)
	rVol_VR_P2s : REAL; (*Volumen VR abhängig von P2s [m3]*)
	rFlow_VR : REAL; (* Differenz Volumen VR [m3/s]*)
	rFlow_VR_TJ : REAL; (* Differenz Volumen VR (TJ filter) [m3/s]*)
	rFlow_GMK : REAL; (* Differenz Volumen GMK [m3/s]*)
	rFlow_GMK_TJ : REAL; (* Differenz Volumen GMK (TJ filter) [m3/s]*)
	rFlow_TJ : REAL; (* Differenz Volumen GMK+VR (TJ filter) [m3/s]*)
	rFlow_TJ_lim : REAL; (* limitiertes Differenz Volumen GMK+VR (TJ filter) [m3/s]*)
	rFlow_L : REAL; (* Soll Volumenstrom ausgehend vom Leanox Soll Druck *)
	rVol_GMK_P2 : REAL; (*Volumen GMK abhängig von P2 [m3]*)
	rFlow_Rot : REAL; (*Ersatzvolumenstrom berechnet aus Rotationsleistung in [Nm3/s]*)
	rCF_VR : REAL; (* Correction Factor Volumenänderung in V-Raum *)
	rVol_VR_208 : REAL; (*208 VR Volumen in [m3]*)
	rVol_VR_312 : REAL; (*312 VR Volumen in [m3]*)
	rVol_VR_316 : REAL; (*316 VR Volumen in [m3]*)
	rVol_VR_320 : REAL; (*320 VR Volumen in [m3]*)
	rVol_VR_412 : REAL; (*412 VR Volumen in [m3]*)
	rVol_VR_416 : REAL; (*416 VR Volumen in [m3]*)
	rVol_VR_420 : REAL; (*420 VR Volumen in [m3]*)
	rVol_VR_424 : REAL; (*424 VR Volumen in [m3]*)
	rVol_VR_612 : REAL; (*612 VR Volumen in [m3]*)
	rVol_VR_616 : REAL; (*616 VR Volumen in [m3]*)
	rVol_VR_620 : REAL; (*620 VR Volumen in [m3]*)
	rVol_VR_624 : REAL; (*624 VR Volumen in [m3]*)
	rV_Act : REAL; (*aktueller Volumenstrom in [m3/h]*)
	rV_DK_ist : REAL;
	rV_DK_soll : REAL;
	rFlow_Gas : REAL; (*aktueller Gasvolumenstrom in [m3/h]*)
	rFlow_Gas_M : REAL;
	rFlow_Gas_M_old : REAL;
	rFlow_Gas_old : REAL;
	rV_UB_ist : REAL;
	rV_UB_soll : REAL;
	ssGrenz : INT; (* turbo suction monitoring limit *)
	ssP2s_l : INT;
	TJ_GasM : ARRAY[0..4] OF BOOL; (* TJ gas flow change error *)
	TJ_GasO : ARRAY[0..4] OF BOOL; (* TJ gas flow maximum error *)
	TON_Monitoring1 : TON;
	TON_Monitoring2 : TON;
	TON_SecondTick : TON; (* second tick timer *)
	xTP_PumpPuls : TP;
	ucCountMax : USINT; (* delay counter for gas flow limits *)
	ucCountMaxM : USINT; (* delay counter for gas flow limits *)
	rFlow_VR_Lo : REAL;
	rFlow_VR_Hi : REAL;
	usordnung : UINT;
	usordnung_f : UINT;
	usordnung_n : UINT;
	usordnung_n_f : UINT;
	usReleaseCnt : UINT;
	xRAMPE_Lambda : RAMPE_R; (* maximum speed of lambda change *)
	xRAMPE_Lmin : RAMPE_R; (* limit speed of change of lmin *)
	xRAMPE_Lmin3 : RAMPE_R; (* limit speed of change of lmin 3 *)
	rEng_N_QC_lim : REAL;
	LCRMovAvgFlt_Eng_N_A : LCRMovAvgFlt;
	LCRMovAvgFlt_Eng_N_B : LCRMovAvgFlt;
	FILTER_R_Eng_N_QC : FILTER_R;
	rTV_QC_lim : REAL;
	rCBV_QC_lim : REAL;
	LCRMovAvgFlt_TV_A : LCRMovAvgFlt;
	LCRMovAvgFlt_TV_B : LCRMovAvgFlt;
	FILTER_R_TV_QC : FILTER_R;
	LCRMovAvgFlt_CBV_A : LCRMovAvgFlt;
	LCRMovAvgFlt_CBV_B : LCRMovAvgFlt;
	FILTER_R_CBV_QC : FILTER_R;
	xLamCorr : lLamCorr;
	xLCRCurve_rLam_Trans_Corr_N : LCRCurveByPoints;
	xLCRCurve_rLam_Trans_Corr_N_tab : ARRAY[0..3] OF lcrCurveByPoints_TabEntry_type;
	xLCRCurve_Dyn_Lambda_LimD : LCRCurveByPoints;
	rDLam_Lim_ManOFF : REAL;
	rT_LambdaFreeze_Max : TIME;
	xTP_LambdaFreeze : TP;
	rT_Lam_Corr_Save : TIME;
	xTP_Lambda_Corr_Disable : TP;
	xTP_Lambda_Freeze_LoadReject : TP;
	bPumpErkennungAktiv : BOOL;
	bSimPID_PID_A_Werte : BOOL; (*Insel: verwende für SimPID Werte aus PID_A*)
	rLam_Trans_Corr_N : REAL;
	rN_Delta : REAL; (* Drehzahlabweichung in [U/min]*)
	rPR_p : REAL;
	rdn_p : REAL;
	xTON_LambdaKorr0 : TON;
	rLam_Trans_Corr_old : REAL; (*old value of transient Lambda correction*)
	rLam_Trans_Corr_DN : REAL; (*transient Lambda correction by speed delta*)
	rLam_Trans_Corr_DP : REAL; (*transient Lambda correction by power delta*)
	l_einst_a_tmp : BOOL;
	bPR_neg : BOOL;
	bPR_pos : BOOL;
	rFlow_LIVC_M : REAL;
	R_TRIG_FPR : R_TRIG;
	TP_Dauer : TP := (0);
	rGasFlowSAVE : REAL;
	rGASObergrenze : REAL;
	rGASObergrenzeM : REAL;
	rGasFlowSAVEM : REAL;
	rGasFlowMSAVE : REAL;
	rGasFlow_Ori : REAL;
	iFPRGasRedOpt : INT;
	rFPRGasRed : REAL;
	tFPRGasRedTime : TIME;
	bFiltInputVolFlow_OWN_Filt : BOOL;
	iT_filt_INPUT_T : USINT;
	iT_filt_INPUT_P : USINT;
	ulGasSprungVoldone : UDINT;
	rGasFlow_ORI : REAL;
	rGasFlowM_ORI : REAL;
	GRMAXPrDiff : GR_MAX;
	GRMAXPrDiff_2 : GR_MAX;
	TPSprung : TP;
	TPSprung_2 : TP;
	TPMin : TP;
	TONTrigger : TON;
	bOld_Island : BOOL;
	bOld_Island2 : BOOL;
	rLamGen2_GCBon : REAL := 0.0;
	rGasFlowGen2_GCBon : REAL := 0.0; (* save Gen2 gas flow during NetP or Island *)
	rGasFlowMGen2_GCBon : REAL := 0.0; (* save Gen2 gas flowM during NetP or Island *)
	xTP_GasFlowGen2_lim_AfterGCBoff : TP; (* Pulse to disable Gen2 gas flow incr. after GCBoff*)
	rTimeGasFlowGen2_lim_AfterGCBoff : REAL := 0.3; (*[s] duration to disable Gen2 gas flow incr. after GCBoff*)
	bPrevStartOk : BOOL := FALSE; (*Check of previous start for gas push function*)
	xF_TRIG_TPSprung : F_TRIG; (* Detect falling edge of gas push *)
	rGasFlow_Old_GrC : REAL; (* Store gas flow when no grid event is detected *)
	rGasFlowM_Old_GrC : REAL; (* Store gas flowM when no grid event is detected *)
	rLamCorr_Enrich_Scale : REAL;
	rLam_Trans_Corr_N_Scale : REAL;
	iLam_Thresh_HiCalVal : UINT; (*[kWh/Nm3]*1000*)
	bGasSprungDone_HiGasDens : BOOL;
	rVolPrc_GT1 : REAL; (*Volume percent of gas type 1 [%] *)
	rCorrFactor_HiGasDens : REAL := 1.0;
	xLCRCurve_Lam_Adapt_Offs : LCRCurveByPoints; (*T6 GEN1 island controller lambda adaption offset map*)
END_VAR
```

### Program Logical/EngineController/FastStart (IEC) - + name is program

- FastStart.st (not readable text: treated as protected, skipped)

#### FastStart.var - Local variables
```iecst
(********************************************************************
 * COPYRIGHT -- INNIO Company
 ********************************************************************
 * Program: FastStart
 * File: FastStart.var
 * Author: 502423184
 * Created: March 03, 2016
 ********************************************************************
 * Local variables of program FastStart
 ********************************************************************)
VAR
	bOM_FastStart_Fail : BOOL;
	bOM_FastStart_Okay : BOOL;
	xTP_OM_FastStart_Okay : TP;
	xTP_OM_FastStart_Fail : TP;
	bFS_IP_Offs_OnlyIdle_Ena : BOOL; (*oldname: rIT_off_start_glob_En2*)
	rP_Set_Unred_Norm_old : REAL;
	rCF_IP_StartOffs_P : REAL; (*correction factor from power deviation*)
	rCA_IP_StartOffs_T : REAL; (*ignition point offset from temperatur lookup table*)
	bFS_IP_Offs_Ena : BOOL; (*oldname: rIT_off_start_glob_En*)
	bFS_IP_Offs_Trip : BOOL; (*oldname: rIT_off_start_glob_Trip*)
	xRamp_IP_StartOffs : RAMPE_R;
	rP_Ramp_FS_Norm : REAL;
	bEng_Dem_EDGE : BOOL;
	rTi_Start : REAL;
	bFS_Req : BOOL;
	bFS_Rdy : BOOL;
	bVFS_Req_Test : BOOL;
	bFS_Req_Test : BOOL;
	rTi_Left : REAL;
	rTi_Target : REAL;
	rTi_Desired : REAL;
	rP_Ramp_UL : REAL;
	bTarget_Hold : BOOL;
	xLCRCByP_IP_Pdev : LCRCurveByPoints;
	xLCRCByP_IP_T3LP : LCRCurveByPoints;
	xLCRCByP_Start_Offs : LCRCurveByPoints;
	bFS_Rel : BOOL;
	xIP_EGTCtr : fIP_EGTCtr;
	rP_Targ_Norm : REAL;
	bIP_EGTCtr_Rel : BOOL;
	xLCRCByP_IP_EGT : LCRCurveByPoints;
	rCA_IP_EGTCtr : REAL;
	bVerrigelung : BOOL := 0;
	bVerrigelung2 : BOOL := 0;
	LCRLimScal_ZZPffs : LCRLimScal;
	LCRLimScal_ZZPffs2 : LCRLimScal;
	TON_ITP : TON;
	LCRScal_StartITOffs : LCRScal;
	bITPStAct : BOOL := 0;
	rT_it_offset : REAL;
	rZZPStart_T_low : REAL;
	rZZPStart_T_high : REAL;
	ucCylinderCount : USINT;
	bForce_FastStartOFF : BOOL := 0; (*TRUE = FASTSTART AUSGESCHALTET*)
	bWait_in_Idle : BOOL;
	rTime_before_SY : REAL;
	rDT_Idle : REAL;
	xTON_NetP : TON;
	bTrigger_GT_SafeDev : BOOL;
	TP_GT_SafeDev : TP;
	TP_110sBlock : TP;
	xTOF_R4VFS : TOF;
	TON_PowerReached : TON;
	tStopBlockFS : TIME := T#30s;
	TP_Stop : TP;
	iSSCount : INT;
	bGEN2_transient : BOOL := 0;
	tDelay_Transient : TIME := T#2s;
	TON_Transient : TON;
	tDelay_stable : TIME := T#5s;
	TOF_Transient : TOF;
	rP_des_lastCyl : REAL;
	RAMPE_R_ITP : RAMPE_R;
	tTP_Verrigelung2 : TIME := T#30s;
	TP_bVerrigelung2 : TP;
	xTOF_MnsOk : TOF;
END_VAR
```

### Program Logical/EngineController/PFPDR (IEC) - + Peak Fire Pressure Detection Run

- PFPDR.st (not readable text: treated as protected, skipped)

#### PFPDR.var - Local variables
```iecst
(********************************************************************
 * COPYRIGHT -- INNIO Company
 ********************************************************************
 * Program: PFPDR
 * File: PFPDR.var
 * Author: 502423184
 * Created: April 15, 2016
 ********************************************************************
 * Local variables of program PFPDR
 ********************************************************************)
VAR
	bStartPFPDR_Man : BOOL;
	bAbortPFPDR_Man : BOOL;
	rCA_Sum_Corr : REAL;
	iCnt_Prof : USINT;
	bBad_Cyl : ARRAY[0..24] OF BOOL;
	bStartPFPDR_Auto : BOOL;
	rCnt_Good_Cyl : REAL;
	rCA_Good_Corr : REAL;
	bPFPDR_new : BOOL;
	iCnt_Cyl : USINT;
	xPFPDR : PFPDR;
	bProf_Corr_Act : BOOL;
END_VAR
VAR CONSTANT
	bDeleteCylArray : ARRAY[0..24] OF BOOL := [25(0)];
	rDeleteCylArray : ARRAY[0..24] OF REAL := [25(0.0)];
END_VAR
VAR
	rCA_PFPDR_ABS_Offs : REAL;
	bLeanox_Man_old : BOOL;
	i : USINT;
	rCA_IP_Prof_Lim : ARRAY[0..24] OF REAL;
	rCA_IP_Prof : ARRAY[0..24] OF REAL;
	xLCRRamp_IP : ARRAY[0..24] OF LCRRamp;
END_VAR
VAR CONSTANT
	YELLOW : INT := 46;
	GREEN : INT := 2;
END_VAR
VAR
	iNum_Disp : USINT;
	iNum_Select : INT;
	bSim : BOOL := 0;
	bSimEGT : BOOL := 0;
	rT_SimEGT : REAL;
END_VAR
VAR CONSTANT
	DeleteData : tPFPDR_Data := (0);
END_VAR
VAR
	Data_Act : tPFPDR_Data := (0);
	Data_Cache : tPFPDR_Data := (0);
	rTi_MaxUp : REAL;
	rTi_MaxDown : REAL;
	rTi_Cnt : REAL;
	rTi_Max : REAL;
	rCA_IP_Prof_Raw : ARRAY[0..24] OF REAL;
	rP_Set_Unred_Norm_Old : REAL;
	bAbortPFPDR_Auto : BOOL;
	xTOF_bMsg2896 : TOF;
	xTOF_bMsg2895 : TOF;
	rRatio : REAL;
	rCA_IP_DR_Prof_Temp : REAL;
	rCA_IP_DR_Min : REAL;
END_VAR
```

### Program Logical/EngineController/ignpoint_EC (IEC) - + timing point calculation

- ignpoint.st (not readable text: treated as protected, skipped)

#### ignpoint.var
```iecst
VAR
	ucCylinderCount : USINT; (* loop counter number of cylinder *)
	rCA_IP_Act_Min : REAL; (* minimum cylinder ignition point *)
	rCA_IP_Act_Min_old : REAL; (* last min. cylinder ignition point *)
	ssTurboySample : INT; (* buffer turbobypass pos. samples *)
	ucSampleCount : USINT; (* sample counter turbobypass pos. *)
	PID_A_IgnTiming : PID_A; (* PID controller timing point *)
	rCA_IP_Rel_Max : REAL; (* current max. allowed delta ZZP *) (* Oldname: ssMaxZZPCyl *)
	rCA_IP_Rel_Min : REAL; (* minimal allowed cyl. timing point *) (* Oldname: ZZPZylMinLimit *)
	slKnockOM : ARRAY[0..24] OF DINT;
	slKnockOH : ARRAY[0..24] OF DINT;
	slKPowerOH : DINT;
	slKPowerOM : DINT;
	ucResetCnt : USINT;
	bPELRedAct : BOOL;
	bKlopfregAkt : BOOL; (*knock control activation bit*)
	rCA_IP_Set_Raw : REAL; (* Oldname: W_ZZPRoh *)
	rCA_IP_Power : REAL; (* Oldname: ssZZPPower *)
	rCA_IP_Knock : REAL; (* Oldname: ssZZPKnock *)
	rCA_IP_CylRed : ARRAY[0..24] OF REAL; (* ZZP-Reduktion *) (* Oldname: ssZZPCylRed *)
	rCA_IP_CylRed_PBC : ARRAY[0..24] OF REAL; (* ZZP-Reduktion durch Glühzünden / Pmax *) (* Oldname: ssZZPCylRedPi *)
	bTimingRedAct : ARRAY[0..24] OF BOOL;
	rCA_Ign_Act_Rel : ARRAY[0..24] OF REAL;
	OpHour_Imp : bh_typ;
	xBH_OpHour : BH;
	xRamp_IP_Glob : RAMPE_R;
	xRamp_IP_CBVOpt : RAMPE_R; (* ramp for timing point reduction *)
	rCA_IP_CBVOpt : REAL;
	xMFB50Contr : MFB50Contr := (0);
	iIdx : USINT;
	bIP_Red_Cyl : ARRAY[0..24] OF BOOL;
	rCA_MFB50_Offs : ARRAY[0..24] OF REAL;
	rCA_IP_Retard_LR_Offset : REAL; (*Offset on ignition timing point to react on load rejection by opening of generator circuit breaker*)
	rCA_IP_Retard_LR : REAL; (*Offset on ignition timing point to react on load rejection by opening of generator circuit breaker*)
	Idle_EngOpState : INT;
	xLCRCByP_IP_P : LCRCurveByPoints;
	rCount_LR : REAL;
	rDelta_LR : REAL;
	bDo_Test : BOOL;
	TON_ParaOK : TON;
	TON_ParaWrite : TON;
	tVerzParaWrite : TIME := T#1110ms;
	rP_CbvOptAct : REAL;
	bTrigASGEN1 : BOOL := FALSE;
	bIgnoreWG_IGP : BOOL := FALSE;
	rCA_IgnP_AvgTmp : REAL;
	TON_F_MMD : TON;
	rF_StartIPRed : REAL; (* Startpoint of IP reduction dependent on nominal frequency *)
	bITP_Offs_F_Act : BOOL := TRUE; (* Bit to activate the frequency dependent ITP reduction function *)
	rCA_ITP_Red_F : REAL; (* ITP offset dependent on engine frequency *)
	rCA_Lim_ITP_Red_F : REAL := 0.0; (* Limited ITP offset dependent on engine frequency *)
	xSCRT_ss : fSCRT_ss; (*Steady State SCR Inlet Temp Ctrl*)
	rCA_IP_SCR_Marg : REAL; (*margin temperature to the limit [degCA]*)
	rCA_IP_SCR_Rel_Lim : REAL; (*SCR Inlet Temperature IP Ctrl - IP Offset limitation [degCA]*)
	rT_EGaTC_Diff : REAL; (*Difference between SCR inlet temperature and its limit [degC]*)
	rCA_IP_T_EGaTC_Off_Rel : REAL; (*IP offset to control SCR inlet temperature [degCA]*)
	xRamp_IP_SCRInTemp : RAMPE_R; (*Ramp for ITP change to control SCR inlet temperature*)
	rCA_Ign_Act_Rel_SCR : REAL; (*SCR Inlet Temperature IP Ctrl - Relative SCR IP for KLS90 [degCA]*)
	rCA_ITP_Red_F_min : REAL := -9.0; (*minimal itp adaption in underfrequency*)
	xLCRCByP_IP_P_HC : LCRCurveByPoints; (* load dependent IP profile for HC interim emission solution *)
	refPoint_IP_P_HC : ARRAY[0..2]OF lcrCurveByPoints_TabEntry_type;
	refPoint_IP_P : ARRAY[0..1]OF lcrCurveByPoints_TabEntry_type;
	rCA_TrStRed_UpLim : REAL; (* highest relative ITP of all cylinders*)
	rCA_TrStRed_Aw : REAL; (* TrStRed function relative ITP feedback *)
	xTON_TrStRed_startupDelay : TON; (* auxiliary TON for TrStRed activation *)
	rP_Norm_TrStRed_act : REAL; (*   TrStRed minimum activation power *)
	bTrStRed_active_Para_Cnd : BOOL; (* auxiliary variable for TrStRed activation *)
	bTrStRed_activePower : BOOL; (* auxiliary variable for TrStRed activation *)
	bTrStRed_active_EngOp_Cnd : BOOL; (* auxiliary variable for TrStRed activation *)
	rCA_upLim_RelITP_TrStRed : REAL; (* actual relative ITP limitation by TrStRed function *)
	xTON_TrStRed_TimeOut : TON; (* timeout timer for TrStRed function *)
	xTOF_TrStRed_PFPDR_dis : TOF; (* TOF for PFPDR disable by TrStRed function *)
	xTOF_TrStRed_hiEGT_dis : TOF; (* TOF for high avg.EGT pw.red. disable / timer extension for high cyl.max.EGT alarm by TrStRed function *)
	xTP_TrStRed_Start : TP;
	xTP_TrStRed_Complete : TP;
	tiTON_TrStRed_startupDelay : TIME;
	rCA_TrStRed_IP_Lim_old : REAL;
	rCA_TrStRed_IP_avg_old : REAL;
	bTrStRed_positiveRamp : BOOL; (* TrStRed positive ramp detection for LXplus steady state loss request *)
	rTrStRedRamp_detectFactor : REAL; (* tolerance factor for TrStRed ramp detection *)
	rCA_TrStRed_LX2reset : REAL; (* TrStRed reset threshold for LXplus steady state loss request *)
	xTON_TrStRed_rampDelay_LX2 : TON; (* TON for TrStRed positive ramp detection for LXplus steady state loss request *)
	xTP_TrStRed_ramp_LX2 : TP;
	xF_Trig_Gen2_IDLE_off : F_TRIG; (* detect negative edge of Gen2 active in IDLE *)
END_VAR
```

### Program Logical/EngineController/leanox_EC (IEC) - + LEANOX controller

- leanoxCyclic.st (not readable text: treated as protected, skipped)

- leanoxInit.st (not readable text: treated as protected, skipped)

#### leanox.var
```iecst
VAR
	bGasChange : BOOL; (* flag for changed gas sort *)
	bStorePoint1 : BOOL; (* flag for store first leanox point *)
	bStorePoint2 : BOOL; (* flag for store second leanox point *)
	bStorePoint3 : BOOL; (* flag for store third leanox point (low load) *)
	bStorePoint1OK : BOOL; (* TRUE=first leanox point stored *)
	bStorePoint2OK : BOOL; (* TRUE=second leanox point stored *)
	bStorePoint3OK : BOOL; (* TRUE=third leanox point (low load) stored *)
	ucGassortOld : USINT; (* last state of gas type *)
	ucGassortPoint1 : USINT; (* gas type at stored point 1 *)
	ucGassortPoint2 : USINT; (* gas type at stored point 2 *)
	ucGassortPoint3 : USINT; (* gas type at stored point 3 (low load) *)
	ucCountPoint : USINT; (* counter for sample averages *)
	rPressLeanoxError : REAL; (* leanox controller deviation [mbar] *)
	slPowerSumm : DINT; (* average sample actual power *)
	slPressw1Summ : DINT; (* average sample boost pressure *)
	rPr_Comp_ChT_mbar : REAL; (* boost press. comp. via mixt. temp. [mbar]*)
	rPr_Comp_IgnP_mbar : REAL; (* boost press. comp. via ITP [mbar]*)
	rN_mp_a : REAL; (* speed point 1 for charge pressure comp. *)
	rN_mp_b : REAL; (* speed point 2 for charge pressure comp. *)
	rN_mp_c : REAL; (* speed point 3 for charge pressure comp. *)
	slSpeedSumm : DINT; (* average sample actual speed *)
	rKK1 : REAL; (* scale point for prop. factor boost [bar rpm / K kW]*)
	rKK2 : REAL; (* scale point for prop. factor boost [bar rpm / K kW]*)
	rKK3 : REAL; (* scale point for prop. factor boost [bar rpm / K kW]*)
	LCRScal_DPressZZP : LCRScal; (* FUB scale ign. tim. point comp. *)
	LCRScal_DPT : LCRScal; (* FUB scale mixture temp. comp. *)
	rScDPressZZP_x : REAL; (* power for charge pressure comp. via ITP [kW] *)
	rScDPT_x : REAL; (* power for charge pressure comp. via charge pressure [kW] *)
	rKK : REAL; (* prop. factor for calc. boost press [bar rpm / K kW]*)
	TON_StartLoxMon : TON; (* FUB delay lenox deviation monitor *)
	bCrossOverOld : BOOL; (* check bit if gas mix. starts/stops *)
	bStorePProz : BOOL; (*FALSE = storage ssp_proz value  *)
	rP_Act_l_mis : REAL; (*rectified power set point in case of misfire*)
	rSpeedCorrFactor : REAL;
	bLambdaOffsetIni : BOOL;
	SimPID_Leanox : SimPID4;
	LCRScal_SyncLambda : LCRScal;
	LCRScal_StartLambda : LCRScal;
	rLam_Start_Offset : REAL;
	LCRCByP_FF_LAMBDA : LCRCurveByPoints;
	rPos_GM_AIT_EOT : REAL; (*Gasmixer position according to Air Intake Temp and Engine Oil Temp*)
	rLam_AIT_EOT : REAL; (*Lambda according to Air Intake Temp and Engine Oil Temp*)
	LCRScal_GMPos_EOT : LCRScal;
	LCRScal_GMPos_AIT : LCRScal;
	LCRScal_Lam_EOT : LCRScal;
	LCRScal_Lam_AIT : LCRScal;
	rTempt2Summ : REAL;
	SimPID4_TV_Opt : SimPID4;
	rN_Act : REAL; (* engine speed for p2´ comp. [1/min] *)
	rLambda_offset : REAL;
	rLambda_sync : REAL;
	rLambda_idle : REAL;
	rT_DevLimit1 : REAL; (*time counter for p2´deviation max. *)
	rT_Leanox : REAL; (*time delay for power reduction *)
	bLeanox_FF_off : BOOL;
	rT_Delay_Idle : REAL;
	rT_Delay_Power : REAL;
	rT_DevLimit2 : REAL;
	rP_Red_Ramp_Norm : REAL;
	rP_PProz_Norm : REAL;
	rP_Red_Ramp_Norm_Up : REAL;
	PID_A_Leanox : PID_A;
	PID_A_Enable : BOOL;
	iCnt_Leanox : INT;
	rCA_Ign_Avg : REAL;
	ucCylIndex : USINT;
	rCA_Ign_Avg_Cnt : REAL;
	rPr_p2s_LLCtr : ARRAY[0..4] OF REAL;
	TON_BPBLIC : TON;
	bBPBLIC_act : BOOL;
	tdelay_Trip : TIME;
	rPr_p2sWindow_SY_LFG : REAL;
	rPr_p2sWindow_hys : REAL;
	rLLCtr_kp : REAL;
	rLLCtr_ki : REAL;
	TON_p2s_SY_LFG : TON;
	rDKOptOffset : REAL;
	bPr_p2sWindow_SY_LFG : BOOL; (*TRUE = SY Freigabe*)
	bUebernahme : BOOL; (*TRUE = LL-Regler läuft*)
	rDKOptOffset_u : REAL;
	bEngine_Start : BOOL := 0; (*Für Idle Mode unterscheidung (Idle bei Motorstart (1) oder Idle nach GCB_ON (0)*)
	TON_rN : TON;
	RAMPE_R_Start_Offset : RAMPE_R;
	boldmode_island : BOOL;
	LCRScal_LD_A : ARRAY[0..4] OF LCRScal; (* FUB scale leanox drift compensation for point 1*)
	LCRScal_LD_B : ARRAY[0..4] OF LCRScal; (* FUB scale leanox drift compensation for point 2*)
	rPr_LD_Delta_A : ARRAY[0..4] OF REAL; (* boost press. comp. leanox drift for point 1 [mbar] *)
	rPr_LD_Delta_B : ARRAY[0..4] OF REAL; (* boost press. comp. leanox drift for point 2 [mbar] *)
	iPr_LD_Delta_SP : INT := 1; (* switching point for adding 1 mbar to leanox parameter [mbar] *)
	i : USINT; (*gas sort*)
	iOpH_LD_old : DINT; (*old value for operating hours*)
	xR_TRIG_ParaOK : R_TRIG; (*initialization of actual operating hours*)
	xTP_LAd : TP; (*time pulse for performed leanox adjustment*)
	xTP_CCC : TP; (*time pulse for performed combustion chamber cleaning*)
	xLamStart : fLamStart := (0);
	RAMPE_R_mis : RAMPE_R;
	TON_LNOxImp : TON;
	tLNOx_verz : TIME := T#40ms;
	bBlockTrigger : BOOL := 0;
	rPr_P2_Dev_Lim_Int : REAL;
	rT_DevLimit1I : REAL;
	rT_LeanoxI : REAL;
	rFactErrorOffs : REAL := 1;
	RPSA7I : BOOL;
	TOF_LOXerrGEN2 : TOF := (0); (*Switch OFF delay at LEANOX power reduction w. GEN2*)
	TON_LOXerrGEN2 : TON; (*Switch ON delay at LEANOX power reduction w. GEN2*)
	rGEN2LeanoxRamp : REAL := 0.005; (*Ramp (decreasing) for Leanox deviation power reduction when using GEN2*)
	rP_GEN2_Red_Ramp_Norm_Up : REAL := 0.0003; (*Ramp (increasing) for Leanox deviation power reduction when using GEN2*)
	FILTER_R_PrP2s_SetGEN2 : FILTER_R;
	iLX2 : INT; (*LX cycle index for running the LX2 task*)
	iLX2sampeTime : INT := 100; (*Threshold for LX cycle index for running the LX2 task*)
	TOF_LX_Adj : TOF; (*Auxiliary TOF for Leanox adjustment confirmation button*)
	bBlockSave : BOOL := 0;
	TP_Block : TP;
	TP_LX2_MapReset : TP;
	TP_LX2_NotActive : TP;
	bLeanox_Active_LX2 : BOOL; (* "Leanox Active" definition for LX2 activation *)
	bLX_Para_adjusted : BOOL; (* Leanox adjustment confirmed *)
	rPr_LX2_Offset_Ctrl : REAL; (* Leanox 2.0 controller offset *)
	rPr_LX2_Offset_BPOC : REAL; (* Leanox 2.0 interpolated BPOC offset gas 1-4 *)
	rPr_LX2_FullOffset : REAL; (* Leanox 2.0 full offset *)
	TOF_LX2ramp_LGM : TOF; (* TOF LX2 ramp for Lambda gradient monitoring interface*)
	TOF_LXadj_LGM : TOF; (* TOF LX adj.confirmation for Lambda gradient monitoring interface*)
	rPr_LX2_offset_old : REAL; (* old value of LX2 offset *)
	rLX2Ramp_detectFactor : REAL := 0.999; (* tolerance factor for LX2 ramp detection *)
	bLX2_negativeRamp : BOOL; (* LX2 negative ramp detection for Lambda gradient monitoring interface *)
	TON_LX2rampDelay_LGM : TON; (* TON for LX2 negative ramp detection for Lambda gradient monitoring interface*)
	rCorr_LX_GR_MIN : REAL := 0.94; (* Minimum value of LEANOX speed compensation factor *)
	rCorr_LX_GR_MAX : REAL := 1.05; (* Maximum value of LEANOX speed compensation factor *)
	rN_Factor_OF_MaxP : REAL; (* Frequency dependend LEANOX speed compensation factor at full load *)
	rN_Factor_OF_MinP : REAL; (* Frequency dependend LEANOX speed compensation factor at half load *)
	xSigScalR_rCorr_LX_GR : xSigScal_R; (* Interpolated LEANOX speed compensation factor *)
	TON_N_GR : TON;
	TON_LX2_startupDelay : TON; (* Auxiliary TON for LX2 activation delay at start-up *)
	bLX2_startupDelay : BOOL; (* start-up delay release condition for LX2 activation *)
	tTOF_LXadj_LGM : TIME; (*Auxiliary timer variable*)
	tTON_LX2rampDelay_LGM : TIME; (*Auxiliary timer variable*)
	tTOF_LX2ramp_LGM : TIME; (*Auxiliary timer variable*)
	xTP_BlockSG_SYLFG : TP; (*block sync after loss of release*)
	xTON_sy_lfg_SG_5s : TON; (*time delay to release sync for BPBLIC*)
	xTON_LX2_Skipfire : TON; (*TON delay for LX2 response in skipfire*)
	tiTON_LX2_Skipfire : TIME; (*Auxiliary timer variable*)
	rPr_P2s_Compensations : REAL; (* LEANOX compensations [bar]*)
	rPr_Demand_PCGT : REAL; (* Prechamber gas pressure for calculation of power reduction [bar(abs)]*)
	rA_Fraction_PCGT : REAL; (* Quadratic coefficient for power reduction calculation PCGT *)
	rB_Fraction_PCGT : REAL; (* Linear coefficient for power reduction calculation PCGT *)
	rC_Fraction_PCGT : REAL; (* Free term for power reduction calculation PCGT *)
	xP_el_PCGT_red_Scal : LCRScal := (0); (* FUB scale prechamber gas pressure *)
	rPr_Demand_GR : REAL; (* Gas rail pressure for calculation of power reduction [bar(abs)]*)
	rA_Fraction_GR : REAL; (* Quadratic coefficient for power reduction calculation GR *)
	rB_Fraction_GR : REAL; (* Linear coefficient for power reduction calculation GR *)
	rC_Fraction_GR : REAL; (* Free term for power reduction calculation GR *)
	xP_el_GR_red_Scal : LCRScal := (0); (* FUB scale gas rail pressure *)
	iLxPoint_P_minDiff : INT; (* Leanox points power reference - minimum distance for warning [kW] *)
	xTON_bSav_LDat_P100_Ena : TON; (*TON delay for enabling HMI saving of Leanox reference point 1*)
	xTON_bSav_LDat_P50_Ena : TON; (*TON delay for enabling HMI saving of Leanox reference point 2*)
	xTON_bSav_LDat_P25_Ena : TON; (*TON delay for enabling HMI saving of Leanox reference point 3*)
	xTOF_LX2_learnStop : TOF; (* TOF delay for removing ext BPOC learn stop signal*)
	tiTOF_LX2_learnStop : TIME; (*Auxiliary timer variable*)
	rLX2_fastRampMult_deact : REAL; (*LX2 ramp multiplier for fast deactivation*)
	xLCRPT1_P_LX2_fast : LCRPT1; (*power filter for LX2 load change detection*)
	xLCRPT1_P_LX2_slow : LCRPT1; (*power filter for LX2 load change detection*)
	rPnorm_filtDiff_LX2: REAL; (*normalized power filters difference for LX2 load change detection [%Pnom/s]*)
	xTON_LX2_MinP : TON; (*TON delay for minimum load detection for LX2*)
	xTOF_LX2_MinP_negStep : TOF; (*TOF delay for load change detection at minimum load for LX2*)
	tiTON_LX2_MinP : TIME; (*Auxiliary timer variable*)
	bLX2_MinP : BOOL; (*minimum load detection for LX2*)
	bLX2_P_negStep : BOOL;  (*load step change detection at minimum load for LX2*)
	xTOF_LX2_deact_LoadReject : TOF; (*TOF delay for LX2 fast deactivation*)
	xTOF_LX2_fastRamp_LoadReject : TOF; (*TOF delay for LX2 fast deactivation*)
	iLX2_P_negRamp : INT; (* counter of negative power gradient detections for LX2 fast deactivation*)
	iLX2_P_negRamp_lim : INT; (* limit counter of consequent negative power gradient detections for LX2 fast deactivation*)
	rP_fastFilt_LX2_old : REAL; (*previous cycle value of filtered power for LX2 load change detection*)
	rPnormFilt_Grad_LX2 : REAL; (*normalized power gradient for LX2 fast deactivation [%Pnom/s]*)
	rPnormFilt_GradSum_LX2 : REAL;
	rPnormFilt_GradAvg_LX2 : REAL;  (*1 second average normalized power gradient for LX2 fast deactivation [%Pnom/s]*)
	iLX2_PnormFilt_GradAvg_loop : INT; (*auxiliary index variable*)
	bLX2_P_negRamp : BOOL;  (*load ramp detection at minimum load for LX2*)
	rPr_P2s_Comp_perH2_HL : REAL; (* Boost pressure offset at half load [mbar] *)
	rPr_P2s_Comp_perH2_FL : REAL; (* Boost pressure offset at full load [mbar] *)
	xSigScalR_P2s_Comp_perH2 : xSigScal_R; (* Interpolated boost pressure compensation factor H2 [bar/%H2] *)
	rPr_P2S_Offset_25PrctH2_HL : REAL; (* Boost pressure offset at 25% H2 content at half load [mbar] *)
	rPr_P2S_Offset_25PrctH2_FL : REAL; (* Boost pressure offset at 25% H2 content at full load [mbar] *)
	xSigScalR_P2s_Comp_25PrctH2 : xSigScal_R; (* Interpolated boost pressure compensation factor H2 [mbar] *)
	rPr_P2s_Comp_perH2 : REAL; (* Boost pressure offset depending on H2 content [mbar] *)
	xRamp_Offs_H2 : RAMPE_R; (* Boost pressure offset ramp *)
	bSteadyState_Loss_H2 : BOOL; (* Deactivate steady state of leanox plus for active lean out *)
	rNOx_set_Delta_H2 : REAL := 5; (* NOx limit to reactivate steady state of leanox plus [ppm] *)
	xTON_LX2_learningEna_startup : TON; (* TON for delayed enabling of LX2 learning component at engine start-up *)
	tiTON_LX2_learningEna_startup : TIME; (* Auxiliary timer variable *)
END_VAR
```

### Program Logical/EngineController/DirAirInj (IEC) - + Direct Air Injection

- DirAirInj.st (not readable text: treated as protected, skipped)
